LIN {X 0,Y 225.817,Z 674.182,A -85,B 0,C 180,E1 6457.381,E2 6457.381} C_VEL
LIN {X 0,Y 214.23,Z 687.655,A -85,B 0,C 180,E1 6455.161,E2 6455.161} C_VEL
LIN {X 0,Y 203.462,Z 699.057,A -85,B 0,C 180,E1 6452.795,E2 6452.795} C_VEL
LIN {X 0,Y 192.684,Z 709.547,A -85,B 0,C 180,E1 6450.053,E2 6450.053} C_VEL
LIN {X 0,Y 181.69,Z 719.435,A -85,B 0,C 180,E1 6446.76,E2 6446.76} C_VEL
LIN {X 0,Y 170.711,Z 728.616,A -85,B 0,C 180,E1 6442.794,E2 6442.794} C_VEL
LIN {X 0,Y 158.871,Z 737.935,A -85,B 0,C 180,E1 6437.414,E2 6437.414} C_VEL
LIN {X 0,Y 147.139,Z 746.59,A -85,B 0,C 180,E1 6430.202,E2 6430.202} C_VEL
LIN {X 0,Y 139.422,Z 752.214,A -85,B 0,C 180,E1 6423.514,E2 6423.514} C_VEL
LIN {X 0,Y 133.904,Z 756.398,A -85,B 0,C 180,E1 6416.613,E2 6416.613} C_VEL
LIN {X 0,Y 130.17,Z 759.571,A -85,B 0,C 180,E1 6409.122,E2 6409.122} C_VEL
LIN {X 0,Y 128.361,Z 761.606,A -85,B 0,C 180,E1 6401.683,E2 6401.683} C_VEL
LIN {X 0,Y 127.961,Z 762.61,A -85,B 0,C 180,E1 6394.93,E2 6394.93} C_VEL
LIN {X 0,Y 128.002,Z 762.852,A -85,B 0,C 180,E1 6388.657,E2 6388.657} C_VEL
LIN {X 0,Y 128.093,Z 762.147,A -85,B 0,C 180,E1 6381.019,E2 6381.019} C_VEL
LIN {X 0,Y 129.629,Z 760.118,A -85,B 0,C 180,E1 6372.495,E2 6372.495} C_VEL
LIN {X 0,Y 129.83,Z 759.905,A -85,B 0,C 180,E1 6371.863,E2 6371.863} C_VEL
LIN {X 0,Y 130.126,Z 758.8,A -85,B 0,C 180,E1 6368.482,E2 6368.482} C_VEL
LIN {X 0,Y 129.362,Z 754.834,A -85,B 0,C 180,E1 6358.995,E2 6358.995} C_VEL
LIN {X 0,Y 130.84,Z 753.309,A -85,B 0,C 180,E1 6356.462,E2 6356.462} C_VEL
LIN {X 0,Y 138.498,Z 748.084,A -85,B 0,C 180,E1 6349.483,E2 6349.483} C_VEL
LIN {X 0,Y 147.503,Z 741.893,A -85,B 0,C 180,E1 6343.512,E2 6343.512} C_VEL
LIN {X 0,Y 157.231,Z 734.942,A -85,B 0,C 180,E1 6338.547,E2 6338.547} C_VEL
LIN {X 0,Y 167.979,Z 726.812,A -85,B 0,C 180,E1 6334.18,E2 6334.18} C_VEL
LIN {X 0,Y 179.579,Z 717.4,A -85,B 0,C 180,E1 6330.354,E2 6330.354} C_VEL
LIN {X 0,Y 194.261,Z 704.416,A -85,B 0,C 180,E1 6326.43,E2 6326.43} C_VEL
LIN {X 0,Y 208.067,Z 690.555,A -85,B 0,C 180,E1 6323.401,E2 6323.401} C_VEL
LIN {X 0,Y 219.406,Z 677.998,A -85,B 0,C 180,E1 6321.278,E2 6321.278} C_VEL
LIN {X 0,Y 230.156,Z 664.84,A -85,B 0,C 180,E1 6319.506,E2 6319.506} C_VEL
LIN {X 0,Y 240.236,Z 651.143,A -85,B 0,C 180,E1 6318.026,E2 6318.026} C_VEL
LIN {X 0,Y 249.892,Z 636.482,A -85,B 0,C 180,E1 6316.744,E2 6316.744} C_VEL
LIN {X 0,Y 260.396,Z 618.414,A -85,B 0,C 180,E1 6315.489,E2 6315.489} C_VEL
LIN {X 0,Y 270.426,Z 597.812,A -85,B 0,C 180,E1 6314.396,E2 6314.396} C_VEL
LIN {X 0,Y 277.33,Z 581.05,A -85,B 0,C 180,E1 6313.706,E2 6313.706} C_VEL
LIN {X 0,Y 283.119,Z 564.422,A -85,B 0,C 180,E1 6313.162,E2 6313.162} C_VEL
LIN {X 0,Y 288.085,Z 547.062,A -85,B 0,C 180,E1 6312.718,E2 6312.718} C_VEL
LIN {X 0,Y 292.005,Z 529.565,A -85,B 0,C 180,E1 6312.361,E2 6312.361} C_VEL
LIN {X 0,Y 294.954,Z 511.261,A -85,B 0,C 180,E1 6312.045,E2 6312.045} C_VEL
LIN {X 0,Y 303.683,Z 432.891,A -85,B 0,C 180,E1 6310.873,E2 6310.873} C_VEL
LIN {X 0,Y 301.535,Z 427.301,A -85,B 0,C 180,E1 6307.622,E2 6307.622} C_VEL
LIN {X 0,Y 300.202,Z 423.933,A -85,B 0,C 180,E1 6304.585,E2 6304.585} C_VEL
LIN {X 0,Y 299.445,Z 421.761,A -85,B 0,C 180,E1 6299.617,E2 6299.617} C_VEL
LIN {X 0,Y 300.396,Z 424.417,A -85,B 0,C 180,E1 6294.557,E2 6294.557} C_VEL
LIN {X 0,Y 301.941,Z 428.499,A -85,B 0,C 180,E1 6291.334,E2 6291.334} C_VEL
LIN {X 0,Y 303.958,Z 433.602,A -85,B 0,C 180,E1 6288.472,E2 6288.472} C_VEL
LIN {X 0,Y 306.454,Z 440.443,A -85,B 0,C 180,E1 6285.691,E2 6285.691} C_VEL
LIN {X 0,Y 309.329,Z 448.867,A -85,B 0,C 180,E1 6283.039,E2 6283.039} C_VEL
LIN {X 0,Y 316.914,Z 468.169,A -85,B 0,C 180,E1 6277.801,E2 6277.801} C_VEL
LIN {X 0,Y 327.353,Z 485.396,A -85,B 0,C 180,E1 6272.829,E2 6272.829} C_VEL
LIN {X 0,Y 339.675,Z 500.381,A -85,B 0,C 180,E1 6268.401,E2 6268.401} C_VEL
LIN {X 0,Y 361.119,Z 520.754,A -85,B 0,C 180,E1 6262.322,E2 6262.322} C_VEL
LIN {X 0,Y 383.771,Z 538.59,A -85,B 0,C 180,E1 6257.155,E2 6257.155} C_VEL
LIN {X 0,Y 393.502,Z 546.007,A -85,B 0,C 180,E1 6254.935,E2 6254.935} C_VEL
LIN {X 0,Y 403.779,Z 553.746,A -85,B 0,C 180,E1 6252.443,E2 6252.443} C_VEL
LIN {X 0,Y 413.394,Z 561.034,A -85,B 0,C 180,E1 6249.938,E2 6249.938} C_VEL
LIN {X 0,Y 423.167,Z 568.574,A -85,B 0,C 180,E1 6247.215,E2 6247.215} C_VEL
LIN {X 0,Y 430.163,Z 573.895,A -85,B 0,C 180,E1 6245.166,E2 6245.166} C_VEL
LIN {X 0,Y 438.79,Z 580.22,A -85,B 0,C 180,E1 6242.527,E2 6242.527} C_VEL
LIN {X 0,Y 446.99,Z 586.446,A -85,B 0,C 180,E1 6239.78,E2 6239.78} C_VEL
LIN {X 0,Y 453.825,Z 591.043,A -85,B 0,C 180,E1 6237.388,E2 6237.388} C_VEL
LIN {X 0,Y 460.622,Z 596.321,A -85,B 0,C 180,E1 6234.765,E2 6234.765} C_VEL
LIN {X 0,Y 467.284,Z 600.659,A -85,B 0,C 180,E1 6231.988,E2 6231.988} C_VEL
LIN {X 0,Y 471.291,Z 603.671,A -85,B 0,C 180,E1 6230.1,E2 6230.1} C_VEL
LIN {X 0,Y 476.325,Z 607.46,A -85,B 0,C 180,E1 6227.466,E2 6227.466} C_VEL
LIN {X 0,Y 480.91,Z 610.202,A -85,B 0,C 180,E1 6224.802,E2 6224.802} C_VEL
LIN {X 0,Y 484.657,Z 612.219,A -85,B 0,C 180,E1 6222.267,E2 6222.267} C_VEL
LIN {X 0,Y 487.465,Z 614.83,A -85,B 0,C 180,E1 6219.682,E2 6219.682} C_VEL
LIN {X 0,Y 489.719,Z 616.73,A -85,B 0,C 180,E1 6217.036,E2 6217.036} C_VEL
LIN {X 0,Y 491.268,Z 617.837,A -85,B 0,C 180,E1 6214.435,E2 6214.435} C_VEL
LIN {X 0,Y 492.185,Z 618.418,A -85,B 0,C 180,E1 6211.779,E2 6211.779} C_VEL
LIN {X 0,Y 492.284,Z 618.462,A -85,B 0,C 180,E1 6209.302,E2 6209.302} C_VEL
LIN {X 0,Y 491.761,Z 618.158,A -85,B 0,C 180,E1 6206.706,E2 6206.706} C_VEL
LIN {X 0,Y 490.502,Z 617.291,A -85,B 0,C 180,E1 6204.151,E2 6204.151} C_VEL
LIN {X 0,Y 488.442,Z 615.733,A -85,B 0,C 180,E1 6201.399,E2 6201.399} C_VEL
LIN {X 0,Y 485.933,Z 613.485,A -85,B 0,C 180,E1 6198.849,E2 6198.849} C_VEL
LIN {X 0,Y 483.548,Z 611.506,A -85,B 0,C 180,E1 6196.893,E2 6196.893} C_VEL
LIN {X 0,Y 479.591,Z 609.49,A -85,B 0,C 180,E1 6194.4,E2 6194.4} C_VEL
LIN {X 0,Y 474.776,Z 606.383,A -85,B 0,C 180,E1 6191.714,E2 6191.714} C_VEL
LIN {X 0,Y 469.767,Z 602.368,A -85,B 0,C 180,E1 6189.133,E2 6189.133} C_VEL
LIN {X 0,Y 464.002,Z 598.659,A -85,B 0,C 180,E1 6186.636,E2 6186.636} C_VEL
LIN {X 0,Y 457.84,Z 594.204,A -85,B 0,C 180,E1 6184.129,E2 6184.129} C_VEL
LIN {X 0,Y 452.424,Z 590.187,A -85,B 0,C 180,E1 6182.133,E2 6182.133} C_VEL
LIN {X 0,Y 445.952,Z 585.668,A -85,B 0,C 180,E1 6179.856,E2 6179.856} C_VEL
LIN {X 0,Y 438.303,Z 579.905,A -85,B 0,C 180,E1 6177.33,E2 6177.33} C_VEL
LIN {X 0,Y 430.019,Z 573.781,A -85,B 0,C 180,E1 6174.79,E2 6174.79} C_VEL
LIN {X 0,Y 422.676,Z 568.214,A -85,B 0,C 180,E1 6172.641,E2 6172.641} C_VEL
LIN {X 0,Y 412.652,Z 560.525,A -85,B 0,C 180,E1 6169.875,E2 6169.875} C_VEL
LIN {X 0,Y 403.258,Z 553.328,A -85,B 0,C 180,E1 6167.428,E2 6167.428} C_VEL
LIN {X 0,Y 392.511,Z 545.225,A -85,B 0,C 180,E1 6164.83,E2 6164.83} C_VEL
LIN {X 0,Y 382.505,Z 537.63,A -85,B 0,C 180,E1 6162.562,E2 6162.562} C_VEL
LIN {X 0,Y 358.465,Z 518.462,A -85,B 0,C 180,E1 6156.999,E2 6156.999} C_VEL
LIN {X 0,Y 337.709,Z 498.182,A -85,B 0,C 180,E1 6150.96,E2 6150.96} C_VEL
LIN {X 0,Y 325.984,Z 483.515,A -85,B 0,C 180,E1 6146.604,E2 6146.604} C_VEL
LIN {X 0,Y 315.507,Z 465.154,A -85,B 0,C 180,E1 6141.374,E2 6141.374} C_VEL
LIN {X 0,Y 307.789,Z 444.262,A -85,B 0,C 180,E1 6135.594,E2 6135.594} C_VEL
LIN {X 0,Y 304.86,Z 435.971,A -85,B 0,C 180,E1 6132.598,E2 6132.598} C_VEL
LIN {X 0,Y 302.482,Z 429.806,A -85,B 0,C 180,E1 6129.514,E2 6129.514} C_VEL
LIN {X 0,Y 301.107,Z 426.479,A -85,B 0,C 180,E1 6127.153,E2 6127.153} C_VEL
LIN {X 0,Y 300.159,Z 423.881,A -85,B 0,C 180,E1 6124.777,E2 6124.777} C_VEL
LIN {X 0,Y 299.447,Z 421.735,A -85,B 0,C 180,E1 6120,E2 6120} C_VEL
LIN {X 0,Y 300.405,Z 424.423,A -85,B 0,C 180,E1 6114.844,E2 6114.844} C_VEL
LIN {X 0,Y 301.897,Z 428.384,A -85,B 0,C 180,E1 6111.716,E2 6111.716} C_VEL
LIN {X 0,Y 303.703,Z 432.989,A -85,B 0,C 180,E1 6109.095,E2 6109.095} C_VEL
LIN {X 0,Y 294.265,Z 516.426,A -85,B 0,C 180,E1 6107.873,E2 6107.873} C_VEL
LIN {X 0,Y 289.898,Z 539.96,A -85,B 0,C 180,E1 6107.438,E2 6107.438} C_VEL
LIN {X 0,Y 284.283,Z 560.709,A -85,B 0,C 180,E1 6106.941,E2 6106.941} C_VEL
LIN {X 0,Y 278.714,Z 577.321,A -85,B 0,C 180,E1 6106.429,E2 6106.429} C_VEL
LIN {X 0,Y 272.26,Z 593.566,A -85,B 0,C 180,E1 6105.794,E2 6105.794} C_VEL
LIN {X 0,Y 264.94,Z 609.422,A -85,B 0,C 180,E1 6105.02,E2 6105.02} C_VEL
LIN {X 0,Y 256.772,Z 624.857,A -85,B 0,C 180,E1 6104.092,E2 6104.092} C_VEL
LIN {X 0,Y 247.786,Z 639.83,A -85,B 0,C 180,E1 6102.986,E2 6102.986} C_VEL
LIN {X 0,Y 237.153,Z 655.552,A -85,B 0,C 180,E1 6101.535,E2 6101.535} C_VEL
LIN {X 0,Y 222.822,Z 674.005,A -85,B 0,C 180,E1 6099.308,E2 6099.308} C_VEL
LIN {X 0,Y 211.394,Z 686.997,A -85,B 0,C 180,E1 6097.253,E2 6097.253} C_VEL
LIN {X 0,Y 199.871,Z 698.879,A -85,B 0,C 180,E1 6094.872,E2 6094.872} C_VEL
LIN {X 0,Y 188.745,Z 709.369,A -85,B 0,C 180,E1 6092.199,E2 6092.199} C_VEL
LIN {X 0,Y 177.345,Z 719.257,A -85,B 0,C 180,E1 6088.967,E2 6088.967} C_VEL
LIN {X 0,Y 166.079,Z 728.293,A -85,B 0,C 180,E1 6085.113,E2 6085.113} C_VEL
LIN {X 0,Y 154.39,Z 737.049,A -85,B 0,C 180,E1 6080.121,E2 6080.121} C_VEL
LIN {X 0,Y 141.499,Z 746.082,A -85,B 0,C 180,E1 6072.7,E2 6072.7} C_VEL
LIN {X 0,Y 132.688,Z 752.036,A -85,B 0,C 180,E1 6065.462,E2 6065.462} C_VEL
LIN {X 0,Y 126.667,Z 756.22,A -85,B 0,C 180,E1 6058.266,E2 6058.266} C_VEL
LIN {X 0,Y 122.584,Z 759.342,A -85,B 0,C 180,E1 6050.53,E2 6050.53} C_VEL
LIN {X 0,Y 120.454,Z 761.429,A -85,B 0,C 180,E1 6042.462,E2 6042.462} C_VEL
LIN {X 0,Y 119.963,Z 762.434,A -85,B 0,C 180,E1 6035.26,E2 6035.26} C_VEL
LIN {X 0,Y 120.001,Z 762.677,A -85,B 0,C 180,E1 6028.568,E2 6028.568} C_VEL
LIN {X 0,Y 120.132,Z 761.97,A -85,B 0,C 180,E1 6020.419,E2 6020.419} C_VEL
LIN {X 0,Y 121.918,Z 759.933,A -85,B 0,C 180,E1 6011.324,E2 6011.324} C_VEL
LIN {X 0,Y 125.803,Z 756.85,A -85,B 0,C 180,E1 6003.065,E2 6003.065} C_VEL
LIN {X 0,Y 130.84,Z 753.309,A -85,B 0,C 180,E1 5996.462,E2 5996.462} C_VEL
LIN {X 0,Y 132.864,Z 751.373,A -85,B 0,C 180,E1 5993.316,E2 5993.316} C_VEL
LIN {X 0,Y 136.774,Z 745.591,A -85,B 0,C 180,E1 5984.772,E2 5984.772} C_VEL
LIN {X 0,Y 139.622,Z 743.303,A -85,B 0,C 180,E1 5982.461,E2 5982.461} C_VEL
LIN {X 0,Y 150.928,Z 735.701,A -85,B 0,C 180,E1 5976.725,E2 5976.725} C_VEL
LIN {X 0,Y 162.074,Z 727.717,A -85,B 0,C 180,E1 5972.319,E2 5972.319} C_VEL
LIN {X 0,Y 173.278,Z 719.078,A -85,B 0,C 180,E1 5968.719,E2 5968.719} C_VEL
LIN {X 0,Y 185.083,Z 709.19,A -85,B 0,C 180,E1 5965.568,E2 5965.568} C_VEL
LIN {X 0,Y 196.552,Z 698.7,A -85,B 0,C 180,E1 5962.979,E2 5962.979} C_VEL
LIN {X 0,Y 208.386,Z 686.819,A -85,B 0,C 180,E1 5960.686,E2 5960.686} C_VEL
LIN {X 0,Y 222.605,Z 670.953,A -85,B 0,C 180,E1 5958.326,E2 5958.326} C_VEL
LIN {X 0,Y 235.611,Z 654.115,A -85,B 0,C 180,E1 5956.469,E2 5956.469} C_VEL
LIN {X 0,Y 245.822,Z 639.217,A -85,B 0,C 180,E1 5955.177,E2 5955.177} C_VEL
LIN {X 0,Y 254.679,Z 624.68,A -85,B 0,C 180,E1 5954.162,E2 5954.162} C_VEL
LIN {X 0,Y 262.974,Z 609.246,A -85,B 0,C 180,E1 5953.285,E2 5953.285} C_VEL
LIN {X 0,Y 270.399,Z 593.389,A -85,B 0,C 180,E1 5952.554,E2 5952.554} C_VEL
LIN {X 0,Y 277.407,Z 575.902,A -85,B 0,C 180,E1 5951.913,E2 5951.913} C_VEL
LIN {X 0,Y 284.639,Z 553.835,A -85,B 0,C 180,E1 5951.303,E2 5951.303} C_VEL
LIN {X 0,Y 289.757,Z 532.601,A -85,B 0,C 180,E1 5950.873,E2 5950.873} C_VEL
LIN {X 0,Y 292.91,Z 514.474,A -85,B 0,C 180,E1 5950.565,E2 5950.565} C_VEL
LIN {X 0,Y 301.601,Z 438.572,A -85,B 0,C 180,E1 5949.445,E2 5949.445} C_VEL
LIN {X 0,Y 300.034,Z 434.394,A -85,B 0,C 180,E1 5946.698,E2 5946.698} C_VEL
LIN {X 0,Y 299.09,Z 431.72,A -85,B 0,C 180,E1 5944.218,E2 5944.218} C_VEL
LIN {X 0,Y 298.467,Z 429.724,A -85,B 0,C 180,E1 5939.616,E2 5939.616} C_VEL
LIN {X 0,Y 299.335,Z 432.351,A -85,B 0,C 180,E1 5934.729,E2 5934.729} C_VEL
LIN {X 0,Y 300.717,Z 436.195,A -85,B 0,C 180,E1 5931.684,E2 5931.684} C_VEL
LIN {X 0,Y 302.598,Z 441.275,A -85,B 0,C 180,E1 5928.854,E2 5928.854} C_VEL
LIN {X 0,Y 304.806,Z 447.733,A -85,B 0,C 180,E1 5926.241,E2 5926.241} C_VEL
LIN {X 0,Y 307.381,Z 455.777,A -85,B 0,C 180,E1 5923.706,E2 5923.706} C_VEL
LIN {X 0,Y 314.649,Z 475.053,A -85,B 0,C 180,E1 5918.418,E2 5918.418} C_VEL
LIN {X 0,Y 324.896,Z 492.411,A -85,B 0,C 180,E1 5913.349,E2 5913.349} C_VEL
LIN {X 0,Y 335.831,Z 506.221,A -85,B 0,C 180,E1 5909.196,E2 5909.196} C_VEL
LIN {X 0,Y 353.843,Z 524.22,A -85,B 0,C 180,E1 5903.7,E2 5903.7} C_VEL
LIN {X 0,Y 379.885,Z 545.436,A -85,B 0,C 180,E1 5897.382,E2 5897.382} C_VEL
LIN {X 0,Y 389.932,Z 553.073,A -85,B 0,C 180,E1 5895.104,E2 5895.104} C_VEL
LIN {X 0,Y 400.416,Z 560.982,A -85,B 0,C 180,E1 5892.553,E2 5892.553} C_VEL
LIN {X 0,Y 410.613,Z 568.64,A -85,B 0,C 180,E1 5889.909,E2 5889.909} C_VEL
LIN {X 0,Y 419.937,Z 575.857,A -85,B 0,C 180,E1 5887.319,E2 5887.319} C_VEL
LIN {X 0,Y 428.263,Z 582.208,A -85,B 0,C 180,E1 5884.885,E2 5884.885} C_VEL
LIN {X 0,Y 436.186,Z 587.913,A -85,B 0,C 180,E1 5882.435,E2 5882.435} C_VEL
LIN {X 0,Y 443.453,Z 593.466,A -85,B 0,C 180,E1 5880.021,E2 5880.021} C_VEL
LIN {X 0,Y 451.356,Z 598.755,A -85,B 0,C 180,E1 5877.291,E2 5877.291} C_VEL
LIN {X 0,Y 458.099,Z 604.069,A -85,B 0,C 180,E1 5874.635,E2 5874.635} C_VEL
LIN {X 0,Y 464.596,Z 608.228,A -85,B 0,C 180,E1 5871.938,E2 5871.938} C_VEL
LIN {X 0,Y 469.631,Z 612.116,A -85,B 0,C 180,E1 5869.525,E2 5869.525} C_VEL
LIN {X 0,Y 474.534,Z 615.637,A -85,B 0,C 180,E1 5866.902,E2 5866.902} C_VEL
LIN {X 0,Y 479.033,Z 618.174,A -85,B 0,C 180,E1 5864.257,E2 5864.257} C_VEL
LIN {X 0,Y 481.979,Z 619.832,A -85,B 0,C 180,E1 5862.215,E2 5862.215} C_VEL
LIN {X 0,Y 484.771,Z 622.412,A -85,B 0,C 180,E1 5859.616,E2 5859.616} C_VEL
LIN {X 0,Y 486.974,Z 624.267,A -85,B 0,C 180,E1 5856.957,E2 5856.957} C_VEL
LIN {X 0,Y 488.51,Z 625.367,A -85,B 0,C 180,E1 5854.343,E2 5854.343} C_VEL
LIN {X 0,Y 489.414,Z 625.923,A -85,B 0,C 180,E1 5851.756,E2 5851.756} C_VEL
LIN {X 0,Y 489.504,Z 625.963,A -85,B 0,C 180,E1 5849.298,E2 5849.298} C_VEL
LIN {X 0,Y 488.977,Z 625.658,A -85,B 0,C 180,E1 5846.718,E2 5846.718} C_VEL
LIN {X 0,Y 487.707,Z 624.783,A -85,B 0,C 180,E1 5844.117,E2 5844.117} C_VEL
LIN {X 0,Y 485.615,Z 623.208,A -85,B 0,C 180,E1 5841.356,E2 5841.356} C_VEL
LIN {X 0,Y 483.115,Z 620.952,A -85,B 0,C 180,E1 5838.783,E2 5838.783} C_VEL
LIN {X 0,Y 480.795,Z 619.019,A -85,B 0,C 180,E1 5836.9,E2 5836.9} C_VEL
LIN {X 0,Y 476.652,Z 616.906,A -85,B 0,C 180,E1 5834.302,E2 5834.302} C_VEL
LIN {X 0,Y 471.906,Z 613.842,A -85,B 0,C 180,E1 5831.666,E2 5831.666} C_VEL
LIN {X 0,Y 466.751,Z 609.74,A -85,B 0,C 180,E1 5829.041,E2 5829.041} C_VEL
LIN {X 0,Y 460.786,Z 605.909,A -85,B 0,C 180,E1 5826.471,E2 5826.471} C_VEL
LIN {X 0,Y 454.378,Z 601.236,A -85,B 0,C 180,E1 5823.875,E2 5823.875} C_VEL
LIN {X 0,Y 449.746,Z 597.783,A -85,B 0,C 180,E1 5822.172,E2 5822.172} C_VEL
LIN {X 0,Y 443.405,Z 593.433,A -85,B 0,C 180,E1 5819.964,E2 5819.964} C_VEL
LIN {X 0,Y 435.55,Z 587.487,A -85,B 0,C 180,E1 5817.356,E2 5817.356} C_VEL
LIN {X 0,Y 426.629,Z 580.931,A -85,B 0,C 180,E1 5814.633,E2 5814.633} C_VEL
LIN {X 0,Y 419.431,Z 575.498,A -85,B 0,C 180,E1 5812.547,E2 5812.547} C_VEL
LIN {X 0,Y 411.112,Z 568.993,A -85,B 0,C 180,E1 5810.225,E2 5810.225} C_VEL
LIN {X 0,Y 400.943,Z 561.405,A -85,B 0,C 180,E1 5807.577,E2 5807.577} C_VEL
LIN {X 0,Y 390.538,Z 553.549,A -85,B 0,C 180,E1 5805.046,E2 5805.046} C_VEL
LIN {X 0,Y 380.193,Z 545.656,A -85,B 0,C 180,E1 5802.678,E2 5802.678} C_VEL
LIN {X 0,Y 353.714,Z 524.102,A -85,B 0,C 180,E1 5796.265,E2 5796.265} C_VEL
LIN {X 0,Y 335.517,Z 505.836,A -85,B 0,C 180,E1 5790.687,E2 5790.687} C_VEL
LIN {X 0,Y 324.222,Z 491.478,A -85,B 0,C 180,E1 5786.365,E2 5786.365} C_VEL
LIN {X 0,Y 313.71,Z 473.008,A -85,B 0,C 180,E1 5781.013,E2 5781.013} C_VEL
LIN {X 0,Y 305.885,Z 450.998,A -85,B 0,C 180,E1 5774.869,E2 5774.869} C_VEL
LIN {X 0,Y 303.192,Z 442.887,A -85,B 0,C 180,E1 5771.895,E2 5771.895} C_VEL
LIN {X 0,Y 300.993,Z 436.928,A -85,B 0,C 180,E1 5768.79,E2 5768.79} C_VEL
LIN {X 0,Y 299.888,Z 434.067,A -85,B 0,C 180,E1 5766.702,E2 5766.702} C_VEL
LIN {X 0,Y 299.115,Z 431.763,A -85,B 0,C 180,E1 5764.602,E2 5764.602} C_VEL
LIN {X 0,Y 298.47,Z 429.691,A -85,B 0,C 180,E1 5760,E2 5760} C_VEL
LIN {X 0,Y 299.343,Z 432.355,A -85,B 0,C 180,E1 5755.018,E2 5755.018} C_VEL
LIN {X 0,Y 300.674,Z 436.079,A -85,B 0,C 180,E1 5752.067,E2 5752.067} C_VEL
LIN {X 0,Y 301.616,Z 438.808,A -85,B 0,C 180,E1 5750.505,E2 5750.505} C_VEL
LIN {X 0,Y 292.661,Z 516.428,A -85,B 0,C 180,E1 5749.405,E2 5749.405} C_VEL
LIN {X 0,Y 288.175,Z 540.116,A -85,B 0,C 180,E1 5748.987,E2 5748.987} C_VEL
LIN {X 0,Y 282.578,Z 560.533,A -85,B 0,C 180,E1 5748.526,E2 5748.526} C_VEL
LIN {X 0,Y 276.939,Z 577.145,A -85,B 0,C 180,E1 5748.046,E2 5748.046} C_VEL
LIN {X 0,Y 270.399,Z 593.39,A -85,B 0,C 180,E1 5747.446,E2 5747.446} C_VEL
LIN {X 0,Y 262.974,Z 609.246,A -85,B 0,C 180,E1 5746.715,E2 5746.715} C_VEL
LIN {X 0,Y 254.68,Z 624.681,A -85,B 0,C 180,E1 5745.837,E2 5745.837} C_VEL
LIN {X 0,Y 245.543,Z 639.653,A -85,B 0,C 180,E1 5744.789,E2 5744.789} C_VEL
LIN {X 0,Y 234.715,Z 655.375,A -85,B 0,C 180,E1 5743.41,E2 5743.41} C_VEL
LIN {X 0,Y 220.085,Z 673.827,A -85,B 0,C 180,E1 5741.285,E2 5741.285} C_VEL
LIN {X 0,Y 208.386,Z 686.82,A -85,B 0,C 180,E1 5739.314,E2 5739.314} C_VEL
LIN {X 0,Y 196.551,Z 698.701,A -85,B 0,C 180,E1 5737.021,E2 5737.021} C_VEL
LIN {X 0,Y 184.676,Z 709.545,A -85,B 0,C 180,E1 5734.332,E2 5734.332} C_VEL
LIN {X 0,Y 172.511,Z 719.697,A -85,B 0,C 180,E1 5731.055,E2 5731.055} C_VEL
LIN {X 0,Y 159.918,Z 729.342,A -85,B 0,C 180,E1 5726.9,E2 5726.9} C_VEL
LIN {X 0,Y 144.46,Z 740.113,A -85,B 0,C 180,E1 5720.191,E2 5720.191} C_VEL
LIN {X 0,Y 133.974,Z 746.902,A -85,B 0,C 180,E1 5713.947,E2 5713.947} C_VEL
LIN {X 0,Y 125.682,Z 752.128,A -85,B 0,C 180,E1 5707.197,E2 5707.197} C_VEL
LIN {X 0,Y 119.221,Z 756.252,A -85,B 0,C 180,E1 5699.654,E2 5699.654} C_VEL
LIN {X 0,Y 114.804,Z 759.314,A -85,B 0,C 180,E1 5691.454,E2 5691.454} C_VEL
LIN {X 0,Y 112.489,Z 761.343,A -85,B 0,C 180,E1 5682.838,E2 5682.838} C_VEL
LIN {X 0,Y 111.964,Z 762.29,A -85,B 0,C 180,E1 5675.123,E2 5675.123} C_VEL
LIN {X 0,Y 112,Z 762.502,A -85,B 0,C 180,E1 5668.465,E2 5668.465} C_VEL
LIN {X 0,Y 112.184,Z 761.794,A -85,B 0,C 180,E1 5659.733,E2 5659.733} C_VEL
LIN {X 0,Y 114.245,Z 759.763,A -85,B 0,C 180,E1 5650.045,E2 5650.045} C_VEL
LIN {X 0,Y 118.613,Z 756.657,A -85,B 0,C 180,E1 5641.249,E2 5641.249} C_VEL
LIN {X 0,Y 124.82,Z 752.671,A -85,B 0,C 180,E1 5633.651,E2 5633.651} C_VEL
LIN {X 0,Y 132.911,Z 747.571,A -85,B 0,C 180,E1 5626.804,E2 5626.804} C_VEL
LIN {X 0,Y 139.622,Z 743.303,A -85,B 0,C 180,E1 5622.461,E2 5622.461} C_VEL
LIN {X 0,Y 143.09,Z 740.557,A -85,B 0,C 180,E1 5619.872,E2 5619.872} C_VEL
LIN {X 0,Y 150.268,Z 733.366,A -85,B 0,C 180,E1 5613.073,E2 5613.073} C_VEL
LIN {X 0,Y 154.478,Z 729.986,A -85,B 0,C 180,E1 5610.975,E2 5610.975} C_VEL
LIN {X 0,Y 167.92,Z 720.137,A -85,B 0,C 180,E1 5606.739,E2 5606.739} C_VEL
LIN {X 0,Y 180.885,Z 709.713,A -85,B 0,C 180,E1 5603.439,E2 5603.439} C_VEL
LIN {X 0,Y 192.665,Z 699.314,A -85,B 0,C 180,E1 5600.927,E2 5600.927} C_VEL
LIN {X 0,Y 203.904,Z 688.42,A -85,B 0,C 180,E1 5598.864,E2 5598.864} C_VEL
LIN {X 0,Y 215.623,Z 675.879,A -85,B 0,C 180,E1 5596.987,E2 5596.987} C_VEL
LIN {X 0,Y 227.078,Z 662.245,A -85,B 0,C 180,E1 5595.38,E2 5595.38} C_VEL
LIN {X 0,Y 240.328,Z 644.448,A -85,B 0,C 180,E1 5593.748,E2 5593.748} C_VEL
LIN {X 0,Y 251.896,Z 626.115,A -85,B 0,C 180,E1 5592.485,E2 5592.485} C_VEL
LIN {X 0,Y 260.772,Z 609.99,A -85,B 0,C 180,E1 5591.61,E2 5591.61} C_VEL
LIN {X 0,Y 268.294,Z 594.275,A -85,B 0,C 180,E1 5590.921,E2 5590.921} C_VEL
LIN {X 0,Y 274.913,Z 578.212,A -85,B 0,C 180,E1 5590.358,E2 5590.358} C_VEL
LIN {X 0,Y 280.616,Z 561.843,A -85,B 0,C 180,E1 5589.906,E2 5589.906} C_VEL
LIN {X 0,Y 285.677,Z 544.056,A -85,B 0,C 180,E1 5589.52,E2 5589.52} C_VEL
LIN {X 0,Y 290.482,Z 521.745,A -85,B 0,C 180,E1 5589.127,E2 5589.127} C_VEL
LIN {X 0,Y 294.809,Z 487.75,A -85,B 0,C 180,E1 5588.645,E2 5588.645} C_VEL
LIN {X 0,Y 299.72,Z 444.504,A -85,B 0,C 180,E1 5588.055,E2 5588.055} C_VEL
LIN {X 0,Y 298.696,Z 441.659,A -85,B 0,C 180,E1 5585.957,E2 5585.957} C_VEL
LIN {X 0,Y 298.05,Z 439.601,A -85,B 0,C 180,E1 5584.04,E2 5584.04} C_VEL
LIN {X 0,Y 297.489,Z 437.69,A -85,B 0,C 180,E1 5579.615,E2 5579.615} C_VEL
LIN {X 0,Y 298.25,Z 440.161,A -85,B 0,C 180,E1 5574.999,E2 5574.999} C_VEL
LIN {X 0,Y 299.554,Z 444.038,A -85,B 0,C 180,E1 5571.941,E2 5571.941} C_VEL
LIN {X 0,Y 301.458,Z 449.556,A -85,B 0,C 180,E1 5568.957,E2 5568.957} C_VEL
LIN {X 0,Y 303.516,Z 456.1,A -85,B 0,C 180,E1 5566.425,E2 5566.425} C_VEL
LIN {X 0,Y 305.808,Z 463.874,A -85,B 0,C 180,E1 5564.059,E2 5564.059} C_VEL
LIN {X 0,Y 312.923,Z 483.011,A -85,B 0,C 180,E1 5558.736,E2 5558.736} C_VEL
LIN {X 0,Y 323.889,Z 501.543,A -85,B 0,C 180,E1 5553.259,E2 5553.259} C_VEL
LIN {X 0,Y 338.433,Z 519.223,A -85,B 0,C 180,E1 5547.772,E2 5547.772} C_VEL
LIN {X 0,Y 357.634,Z 537.531,A -85,B 0,C 180,E1 5542.042,E2 5542.042} C_VEL
LIN {X 0,Y 380.681,Z 555.751,A -85,B 0,C 180,E1 5536.515,E2 5536.515} C_VEL
LIN {X 0,Y 391.612,Z 564.172,A -85,B 0,C 180,E1 5533.944,E2 5533.944} C_VEL
LIN {X 0,Y 401.536,Z 571.781,A -85,B 0,C 180,E1 5531.449,E2 5531.449} C_VEL
LIN {X 0,Y 410.626,Z 578.592,A -85,B 0,C 180,E1 5529.033,E2 5529.033} C_VEL
LIN {X 0,Y 419.479,Z 585.163,A -85,B 0,C 180,E1 5526.554,E2 5526.554} C_VEL
LIN {X 0,Y 428.549,Z 592.2,A -85,B 0,C 180,E1 5523.837,E2 5523.837} C_VEL
LIN {X 0,Y 436.065,Z 597.592,A -85,B 0,C 180,E1 5521.461,E2 5521.461} C_VEL
LIN {X 0,Y 442.945,Z 602.736,A -85,B 0,C 180,E1 5519.12,E2 5519.12} C_VEL
LIN {X 0,Y 449.61,Z 607.3,A -85,B 0,C 180,E1 5516.774,E2 5516.774} C_VEL
LIN {X 0,Y 456.445,Z 612.475,A -85,B 0,C 180,E1 5514.041,E2 5514.041} C_VEL
LIN {X 0,Y 463.052,Z 616.623,A -85,B 0,C 180,E1 5511.267,E2 5511.267} C_VEL
LIN {X 0,Y 468.396,Z 620.937,A -85,B 0,C 180,E1 5508.544,E2 5508.544} C_VEL
LIN {X 0,Y 473.356,Z 624.177,A -85,B 0,C 180,E1 5505.81,E2 5505.81} C_VEL
LIN {X 0,Y 477.617,Z 626.357,A -85,B 0,C 180,E1 5503.189,E2 5503.189} C_VEL
LIN {X 0,Y 479.81,Z 628.141,A -85,B 0,C 180,E1 5501.417,E2 5501.417} C_VEL
LIN {X 0,Y 482.399,Z 630.472,A -85,B 0,C 180,E1 5498.822,E2 5498.822} C_VEL
LIN {X 0,Y 484.472,Z 632.055,A -85,B 0,C 180,E1 5496.16,E2 5496.16} C_VEL
LIN {X 0,Y 485.834,Z 633.014,A -85,B 0,C 180,E1 5493.46,E2 5493.46} C_VEL
LIN {X 0,Y 486.4,Z 633.343,A -85,B 0,C 180,E1 5490.942,E2 5490.942} C_VEL
LIN {X 0,Y 486.324,Z 633.313,A -85,B 0,C 180,E1 5488.351,E2 5488.351} C_VEL
LIN {X 0,Y 485.442,Z 632.747,A -85,B 0,C 180,E1 5485.63,E2 5485.63} C_VEL
LIN {X 0,Y 483.881,Z 631.639,A -85,B 0,C 180,E1 5482.998,E2 5482.998} C_VEL
LIN {X 0,Y 481.607,Z 629.742,A -85,B 0,C 180,E1 5480.32,E2 5480.32} C_VEL
LIN {X 0,Y 478.826,Z 627.154,A -85,B 0,C 180,E1 5477.704,E2 5477.704} C_VEL
LIN {X 0,Y 475.145,Z 625.14,A -85,B 0,C 180,E1 5475.25,E2 5475.25} C_VEL
LIN {X 0,Y 470.438,Z 622.377,A -85,B 0,C 180,E1 5472.564,E2 5472.564} C_VEL
LIN {X 0,Y 465.099,Z 618.372,A -85,B 0,C 180,E1 5469.752,E2 5469.752} C_VEL
LIN {X 0,Y 461.325,Z 615.512,A -85,B 0,C 180,E1 5467.981,E2 5467.981} C_VEL
LIN {X 0,Y 454.716,Z 611.271,A -85,B 0,C 180,E1 5465.253,E2 5465.253} C_VEL
LIN {X 0,Y 448.032,Z 606.006,A -85,B 0,C 180,E1 5462.634,E2 5462.634} C_VEL
LIN {X 0,Y 439.737,Z 600.437,A -85,B 0,C 180,E1 5459.776,E2 5459.776} C_VEL
LIN {X 0,Y 432.331,Z 594.826,A -85,B 0,C 180,E1 5457.337,E2 5457.337} C_VEL
LIN {X 0,Y 423.676,Z 588.509,A -85,B 0,C 180,E1 5454.681,E2 5454.681} C_VEL
LIN {X 0,Y 415.058,Z 582.011,A -85,B 0,C 180,E1 5452.201,E2 5452.201} C_VEL
LIN {X 0,Y 406.119,Z 575.128,A -85,B 0,C 180,E1 5449.751,E2 5449.751} C_VEL
LIN {X 0,Y 396.371,Z 567.744,A -85,B 0,C 180,E1 5447.23,E2 5447.23} C_VEL
LIN {X 0,Y 385.645,Z 559.667,A -85,B 0,C 180,E1 5444.64,E2 5444.64} C_VEL
LIN {X 0,Y 376.001,Z 552.329,A -85,B 0,C 180,E1 5442.438,E2 5442.438} C_VEL
LIN {X 0,Y 351.631,Z 532.3,A -85,B 0,C 180,E1 5436.312,E2 5436.312} C_VEL
LIN {X 0,Y 332.627,Z 512.698,A -85,B 0,C 180,E1 5430.183,E2 5430.183} C_VEL
LIN {X 0,Y 321.436,Z 497.955,A -85,B 0,C 180,E1 5425.669,E2 5425.669} C_VEL
LIN {X 0,Y 311.111,Z 478.937,A -85,B 0,C 180,E1 5420.114,E2 5420.114} C_VEL
LIN {X 0,Y 304.032,Z 457.731,A -85,B 0,C 180,E1 5414.134,E2 5414.134} C_VEL
LIN {X 0,Y 301.637,Z 450.053,A -85,B 0,C 180,E1 5411.278,E2 5411.278} C_VEL
LIN {X 0,Y 299.605,Z 444.184,A -85,B 0,C 180,E1 5408.154,E2 5408.154} C_VEL
LIN {X 0,Y 298.535,Z 441.209,A -85,B 0,C 180,E1 5405.863,E2 5405.863} C_VEL
LIN {X 0,Y 298.013,Z 439.549,A -85,B 0,C 180,E1 5404.233,E2 5404.233} C_VEL
LIN {X 0,Y 297.493,Z 437.65,A -85,B 0,C 180,E1 5400,E2 5400} C_VEL
LIN {X 0,Y 298.257,Z 440.165,A -85,B 0,C 180,E1 5395.289,E2 5395.289} C_VEL
LIN {X 0,Y 299.512,Z 443.922,A -85,B 0,C 180,E1 5392.326,E2 5392.326} C_VEL
LIN {X 0,Y 299.699,Z 444.754,A -85,B 0,C 180,E1 5391.933,E2 5391.933} C_VEL
LIN {X 0,Y 291.267,Z 516.442,A -85,B 0,C 180,E1 5390.953,E2 5390.953} C_VEL
LIN {X 0,Y 286.632,Z 540.398,A -85,B 0,C 180,E1 5390.551,E2 5390.551} C_VEL
LIN {X 0,Y 281.092,Z 560.358,A -85,B 0,C 180,E1 5390.129,E2 5390.129} C_VEL
LIN {X 0,Y 275.387,Z 576.97,A -85,B 0,C 180,E1 5389.681,E2 5389.681} C_VEL
LIN {X 0,Y 268.766,Z 593.214,A -85,B 0,C 180,E1 5389.12,E2 5389.12} C_VEL
LIN {X 0,Y 261.241,Z 609.07,A -85,B 0,C 180,E1 5388.434,E2 5388.434} C_VEL
LIN {X 0,Y 252.827,Z 624.505,A -85,B 0,C 180,E1 5387.61,E2 5387.61} C_VEL
LIN {X 0,Y 243.548,Z 639.477,A -85,B 0,C 180,E1 5386.624,E2 5386.624} C_VEL
LIN {X 0,Y 232.242,Z 655.6,A -85,B 0,C 180,E1 5385.284,E2 5385.284} C_VEL
LIN {X 0,Y 217.618,Z 673.65,A -85,B 0,C 180,E1 5383.308,E2 5383.308} C_VEL
LIN {X 0,Y 205.655,Z 686.642,A -85,B 0,C 180,E1 5381.433,E2 5381.433} C_VEL
LIN {X 0,Y 193.519,Z 698.523,A -85,B 0,C 180,E1 5379.241,E2 5379.241} C_VEL
LIN {X 0,Y 181.713,Z 709.012,A -85,B 0,C 180,E1 5376.751,E2 5376.751} C_VEL
LIN {X 0,Y 169.507,Z 718.9,A -85,B 0,C 180,E1 5373.701,E2 5373.701} C_VEL
LIN {X 0,Y 157.102,Z 728.08,A -85,B 0,C 180,E1 5369.936,E2 5369.936} C_VEL
LIN {X 0,Y 143.358,Z 737.436,A -85,B 0,C 180,E1 5364.626,E2 5364.626} C_VEL
LIN {X 0,Y 129.372,Z 746.054,A -85,B 0,C 180,E1 5357.234,E2 5357.234} C_VEL
LIN {X 0,Y 119.75,Z 751.678,A -85,B 0,C 180,E1 5350.004,E2 5350.004} C_VEL
LIN {X 0,Y 112.564,Z 755.863,A -85,B 0,C 180,E1 5342.201,E2 5342.201} C_VEL
LIN {X 0,Y 107.506,Z 758.986,A -85,B 0,C 180,E1 5333.57,E2 5333.57} C_VEL
LIN {X 0,Y 104.713,Z 761.076,A -85,B 0,C 180,E1 5324.373,E2 5324.373} C_VEL
LIN {X 0,Y 103.978,Z 762.083,A -85,B 0,C 180,E1 5316.071,E2 5316.071} C_VEL
LIN {X 0,Y 104.01,Z 762.355,A -85,B 0,C 180,E1 5308.87,E2 5308.87} C_VEL
LIN {X 0,Y 104.197,Z 761.708,A -85,B 0,C 180,E1 5299.496,E2 5299.496} C_VEL
LIN {X 0,Y 106.644,Z 759.585,A -85,B 0,C 180,E1 5288.555,E2 5288.555} C_VEL
LIN {X 0,Y 111.51,Z 756.493,A -85,B 0,C 180,E1 5279.267,E2 5279.267} C_VEL
LIN {X 0,Y 118.338,Z 752.492,A -85,B 0,C 180,E1 5271.305,E2 5271.305} C_VEL
LIN {X 0,Y 127.072,Z 747.392,A -85,B 0,C 180,E1 5264.279,E2 5264.279} C_VEL
LIN {X 0,Y 137.4,Z 741.135,A -85,B 0,C 180,E1 5258.202,E2 5258.202} C_VEL
LIN {X 0,Y 149.021,Z 733.647,A -85,B 0,C 180,E1 5253.007,E2 5253.007} C_VEL
LIN {X 0,Y 154.478,Z 729.986,A -85,B 0,C 180,E1 5250.975,E2 5250.975} C_VEL
LIN {X 0,Y 158.847,Z 726.473,A -85,B 0,C 180,E1 5249.006,E2 5249.006} C_VEL
LIN {X 0,Y 168.347,Z 717.551,A -85,B 0,C 180,E1 5243.627,E2 5243.627} C_VEL
LIN {X 0,Y 173.066,Z 713.456,A -85,B 0,C 180,E1 5242.084,E2 5242.084} C_VEL
LIN {X 0,Y 188.161,Z 700.718,A -85,B 0,C 180,E1 5238.957,E2 5238.957} C_VEL
LIN {X 0,Y 200.635,Z 689.027,A -85,B 0,C 180,E1 5236.801,E2 5236.801} C_VEL
LIN {X 0,Y 212.242,Z 676.966,A -85,B 0,C 180,E1 5235.063,E2 5235.063} C_VEL
LIN {X 0,Y 223.221,Z 664.309,A -85,B 0,C 180,E1 5233.618,E2 5233.618} C_VEL
LIN {X 0,Y 233.915,Z 650.55,A -85,B 0,C 180,E1 5232.36,E2 5232.36} C_VEL
LIN {X 0,Y 244.153,Z 635.748,A -85,B 0,C 180,E1 5231.275,E2 5231.275} C_VEL
LIN {X 0,Y 255.479,Z 617.08,A -85,B 0,C 180,E1 5230.204,E2 5230.204} C_VEL
LIN {X 0,Y 265.457,Z 597.284,A -85,B 0,C 180,E1 5229.343,E2 5229.343} C_VEL
LIN {X 0,Y 272.626,Z 580.523,A -85,B 0,C 180,E1 5228.777,E2 5228.777} C_VEL
LIN {X 0,Y 278.625,Z 563.896,A -85,B 0,C 180,E1 5228.336,E2 5228.336} C_VEL
LIN {X 0,Y 283.759,Z 546.544,A -85,B 0,C 180,E1 5227.975,E2 5227.975} C_VEL
LIN {X 0,Y 287.792,Z 529.155,A -85,B 0,C 180,E1 5227.679,E2 5227.679} C_VEL
LIN {X 0,Y 290.857,Z 510.941,A -85,B 0,C 180,E1 5227.409,E2 5227.409} C_VEL
LIN {X 0,Y 297.986,Z 450.482,A -85,B 0,C 180,E1 5226.604,E2 5226.604} C_VEL
LIN {X 0,Y 297.013,Z 447.483,A -85,B 0,C 180,E1 5223.861,E2 5223.861} C_VEL
LIN {X 0,Y 296.51,Z 445.66,A -85,B 0,C 180,E1 5219.614,E2 5219.614} C_VEL
LIN {X 0,Y 297.171,Z 447.971,A -85,B 0,C 180,E1 5215.272,E2 5215.272} C_VEL
LIN {X 0,Y 298.349,Z 451.732,A -85,B 0,C 180,E1 5212.296,E2 5212.296} C_VEL
LIN {X 0,Y 300.218,Z 457.515,A -85,B 0,C 180,E1 5209.202,E2 5209.202} C_VEL
LIN {X 0,Y 302.515,Z 465.463,A -85,B 0,C 180,E1 5206.282,E2 5206.282} C_VEL
LIN {X 0,Y 310.925,Z 490.348,A -85,B 0,C 180,E1 5199.234,E2 5199.234} C_VEL
LIN {X 0,Y 320.466,Z 507.275,A -85,B 0,C 180,E1 5194.149,E2 5194.149} C_VEL
LIN {X 0,Y 331.055,Z 521.373,A -85,B 0,C 180,E1 5189.734,E2 5189.734} C_VEL
LIN {X 0,Y 349.886,Z 540.881,A -85,B 0,C 180,E1 5183.478,E2 5183.478} C_VEL
LIN {X 0,Y 374.602,Z 561.138,A -85,B 0,C 180,E1 5177.106,E2 5177.106} C_VEL
LIN {X 0,Y 385.705,Z 569.643,A -85,B 0,C 180,E1 5174.528,E2 5174.528} C_VEL
LIN {X 0,Y 394.75,Z 576.503,A -85,B 0,C 180,E1 5172.3,E2 5172.3} C_VEL
LIN {X 0,Y 405.018,Z 584.149,A -85,B 0,C 180,E1 5169.623,E2 5169.623} C_VEL
LIN {X 0,Y 413.441,Z 590.602,A -85,B 0,C 180,E1 5167.281,E2 5167.281} C_VEL
LIN {X 0,Y 420.229,Z 595.799,A -85,B 0,C 180,E1 5165.3,E2 5165.3} C_VEL
LIN {X 0,Y 428.387,Z 601.723,A -85,B 0,C 180,E1 5162.831,E2 5162.831} C_VEL
LIN {X 0,Y 436.334,Z 607.697,A -85,B 0,C 180,E1 5160.24,E2 5160.24} C_VEL
LIN {X 0,Y 445.139,Z 613.695,A -85,B 0,C 180,E1 5157.188,E2 5157.188} C_VEL
LIN {X 0,Y 452.244,Z 619.182,A -85,B 0,C 180,E1 5154.368,E2 5154.368} C_VEL
LIN {X 0,Y 458.611,Z 623.134,A -85,B 0,C 180,E1 5151.752,E2 5151.752} C_VEL
LIN {X 0,Y 464.442,Z 627.782,A -85,B 0,C 180,E1 5148.838,E2 5148.838} C_VEL
LIN {X 0,Y 469.572,Z 631.192,A -85,B 0,C 180,E1 5146.068,E2 5146.068} C_VEL
LIN {X 0,Y 473.698,Z 633.36,A -85,B 0,C 180,E1 5143.549,E2 5143.549} C_VEL
LIN {X 0,Y 475.746,Z 634.747,A -85,B 0,C 180,E1 5142.008,E2 5142.008} C_VEL
LIN {X 0,Y 478.592,Z 637.36,A -85,B 0,C 180,E1 5139.256,E2 5139.256} C_VEL
LIN {X 0,Y 480.766,Z 639.092,A -85,B 0,C 180,E1 5136.567,E2 5136.567} C_VEL
LIN {X 0,Y 482.099,Z 640.052,A -85,B 0,C 180,E1 5134.162,E2 5134.162} C_VEL
LIN {X 0,Y 482.947,Z 640.557,A -85,B 0,C 180,E1 5131.661,E2 5131.661} C_VEL
LIN {X 0,Y 483.038,Z 640.594,A -85,B 0,C 180,E1 5129.288,E2 5129.288} C_VEL
LIN {X 0,Y 482.483,Z 640.276,A -85,B 0,C 180,E1 5126.674,E2 5126.674} C_VEL
LIN {X 0,Y 481.194,Z 639.383,A -85,B 0,C 180,E1 5124.037,E2 5124.037} C_VEL
LIN {X 0,Y 479.124,Z 637.842,A -85,B 0,C 180,E1 5121.359,E2 5121.359} C_VEL
LIN {X 0,Y 476.58,Z 635.562,A -85,B 0,C 180,E1 5118.75,E2 5118.75} C_VEL
LIN {X 0,Y 474.269,Z 633.623,A -85,B 0,C 180,E1 5116.841,E2 5116.841} C_VEL
LIN {X 0,Y 470.015,Z 631.449,A -85,B 0,C 180,E1 5114.201,E2 5114.201} C_VEL
LIN {X 0,Y 464.998,Z 628.188,A -85,B 0,C 180,E1 5111.446,E2 5111.446} C_VEL
LIN {X 0,Y 459.473,Z 623.751,A -85,B 0,C 180,E1 5108.655,E2 5108.655} C_VEL
LIN {X 0,Y 453.151,Z 619.8,A -85,B 0,C 180,E1 5105.994,E2 5105.994} C_VEL
LIN {X 0,Y 446.02,Z 614.434,A -85,B 0,C 180,E1 5103.156,E2 5103.156} C_VEL
LIN {X 0,Y 439.05,Z 609.666,A -85,B 0,C 180,E1 5100.721,E2 5100.721} C_VEL
LIN {X 0,Y 433.037,Z 605.203,A -85,B 0,C 180,E1 5098.687,E2 5098.687} C_VEL
LIN {X 0,Y 427.855,Z 601.372,A -85,B 0,C 180,E1 5097.013,E2 5097.013} C_VEL
LIN {X 0,Y 420.152,Z 595.736,A -85,B 0,C 180,E1 5094.675,E2 5094.675} C_VEL
LIN {X 0,Y 412.958,Z 590.256,A -85,B 0,C 180,E1 5092.578,E2 5092.578} C_VEL
LIN {X 0,Y 402.495,Z 582.258,A -85,B 0,C 180,E1 5089.699,E2 5089.699} C_VEL
LIN {X 0,Y 393.165,Z 575.258,A -85,B 0,C 180,E1 5087.306,E2 5087.306} C_VEL
LIN {X 0,Y 384.067,Z 568.41,A -85,B 0,C 180,E1 5085.083,E2 5085.083} C_VEL
LIN {X 0,Y 373.47,Z 560.303,A -85,B 0,C 180,E1 5082.638,E2 5082.638} C_VEL
LIN {X 0,Y 348.787,Z 539.862,A -85,B 0,C 180,E1 5076.196,E2 5076.196} C_VEL
LIN {X 0,Y 330.385,Z 520.551,A -85,B 0,C 180,E1 5070.008,E2 5070.008} C_VEL
LIN {X 0,Y 320.31,Z 506.996,A -85,B 0,C 180,E1 5065.765,E2 5065.765} C_VEL
LIN {X 0,Y 310.714,Z 489.893,A -85,B 0,C 180,E1 5060.633,E2 5060.633} C_VEL
LIN {X 0,Y 303.881,Z 470.608,A -85,B 0,C 180,E1 5055.213,E2 5055.213} C_VEL
LIN {X 0,Y 301.788,Z 462.981,A -85,B 0,C 180,E1 5052.874,E2 5052.874} C_VEL
LIN {X 0,Y 299.952,Z 456.715,A -85,B 0,C 180,E1 5050.419,E2 5050.419} C_VEL
LIN {X 0,Y 298.302,Z 451.583,A -85,B 0,C 180,E1 5047.608,E2 5047.608} C_VEL
LIN {X 0,Y 297.098,Z 447.621,A -85,B 0,C 180,E1 5044.439,E2 5044.439} C_VEL
LIN {X 0,Y 296.515,Z 445.614,A -85,B 0,C 180,E1 5040,E2 5040} C_VEL
LIN {X 0,Y 297.178,Z 447.974,A -85,B 0,C 180,E1 5035.562,E2 5035.562} C_VEL
LIN {X 0,Y 297.977,Z 450.647,A -85,B 0,C 180,E1 5033.378,E2 5033.378} C_VEL
LIN {X 0,Y 290.092,Z 516.419,A -85,B 0,C 180,E1 5032.515,E2 5032.515} C_VEL
LIN {X 0,Y 285.335,Z 540.566,A -85,B 0,C 180,E1 5032.132,E2 5032.132} C_VEL
LIN {X 0,Y 279.828,Z 560.183,A -85,B 0,C 180,E1 5031.748,E2 5031.748} C_VEL
LIN {X 0,Y 274.062,Z 576.794,A -85,B 0,C 180,E1 5031.334,E2 5031.334} C_VEL
LIN {X 0,Y 267.364,Z 593.038,A -85,B 0,C 180,E1 5030.813,E2 5030.813} C_VEL
LIN {X 0,Y 259.747,Z 608.894,A -85,B 0,C 180,E1 5030.174,E2 5030.174} C_VEL
LIN {X 0,Y 251.22,Z 624.328,A -85,B 0,C 180,E1 5029.407,E2 5029.407} C_VEL
LIN {X 0,Y 241.807,Z 639.3,A -85,B 0,C 180,E1 5028.486,E2 5028.486} C_VEL
LIN {X 0,Y 230.616,Z 655.021,A -85,B 0,C 180,E1 5027.267,E2 5027.267} C_VEL
LIN {X 0,Y 215.428,Z 673.473,A -85,B 0,C 180,E1 5025.375,E2 5025.375} C_VEL
LIN {X 0,Y 203.214,Z 686.464,A -85,B 0,C 180,E1 5023.606,E2 5023.606} C_VEL
LIN {X 0,Y 190.786,Z 698.345,A -85,B 0,C 180,E1 5021.527,E2 5021.527} C_VEL
LIN {X 0,Y 178.653,Z 708.834,A -85,B 0,C 180,E1 5019.154,E2 5019.154} C_VEL
LIN {X 0,Y 165.862,Z 718.865,A -85,B 0,C 180,E1 5016.177,E2 5016.177} C_VEL
LIN {X 0,Y 153.172,Z 727.901,A -85,B 0,C 180,E1 5012.582,E2 5012.582} C_VEL
LIN {X 0,Y 138.84,Z 737.22,A -85,B 0,C 180,E1 5007.404,E2 5007.404} C_VEL
LIN {X 0,Y 123.963,Z 745.875,A -85,B 0,C 180,E1 5000.011,E2 5000.011} C_VEL
LIN {X 0,Y 113.61,Z 751.5,A -85,B 0,C 180,E1 4992.655,E2 4992.655} C_VEL
LIN {X 0,Y 105.751,Z 755.685,A -85,B 0,C 180,E1 4984.557,E2 4984.557} C_VEL
LIN {X 0,Y 100.102,Z 758.808,A -85,B 0,C 180,E1 4975.433,E2 4975.433} C_VEL
LIN {X 0,Y 96.892,Z 760.899,A -85,B 0,C 180,E1 4965.561,E2 4965.561} C_VEL
LIN {X 0,Y 95.976,Z 761.939,A -85,B 0,C 180,E1 4955.979,E2 4955.979} C_VEL
LIN {X 0,Y 96.009,Z 762.182,A -85,B 0,C 180,E1 4948.807,E2 4948.807} C_VEL
LIN {X 0,Y 96.271,Z 761.531,A -85,B 0,C 180,E1 4938.62,E2 4938.62} C_VEL
LIN {X 0,Y 99.124,Z 759.408,A -85,B 0,C 180,E1 4926.837,E2 4926.837} C_VEL
LIN {X 0,Y 104.582,Z 756.315,A -85,B 0,C 180,E1 4916.983,E2 4916.983} C_VEL
LIN {X 0,Y 112.076,Z 752.314,A -85,B 0,C 180,E1 4908.692,E2 4908.692} C_VEL
LIN {X 0,Y 121.504,Z 747.213,A -85,B 0,C 180,E1 4901.517,E2 4901.517} C_VEL
LIN {X 0,Y 132.497,Z 740.956,A -85,B 0,C 180,E1 4895.421,E2 4895.421} C_VEL
LIN {X 0,Y 144.768,Z 733.445,A -85,B 0,C 180,E1 4890.279,E2 4890.279} C_VEL
LIN {X 0,Y 160.344,Z 723.024,A -85,B 0,C 180,E1 4885.3,E2 4885.3} C_VEL
LIN {X 0,Y 173.066,Z 713.456,A -85,B 0,C 180,E1 4882.084,E2 4882.084} C_VEL
LIN {X 0,Y 177.816,Z 709.254,A -85,B 0,C 180,E1 4880.642,E2 4880.642} C_VEL
LIN {X 0,Y 188.394,Z 698.519,A -85,B 0,C 180,E1 4876.465,E2 4876.465} C_VEL
LIN {X 0,Y 193.333,Z 693.806,A -85,B 0,C 180,E1 4875.333,E2 4875.333} C_VEL
LIN {X 0,Y 208.431,Z 678.786,A -85,B 0,C 180,E1 4873.169,E2 4873.169} C_VEL
LIN {X 0,Y 220.518,Z 665.252,A -85,B 0,C 180,E1 4871.687,E2 4871.687} C_VEL
LIN {X 0,Y 231.327,Z 651.696,A -85,B 0,C 180,E1 4870.513,E2 4870.513} C_VEL
LIN {X 0,Y 241.276,Z 637.702,A -85,B 0,C 180,E1 4869.537,E2 4869.537} C_VEL
LIN {X 0,Y 250.416,Z 623.221,A -85,B 0,C 180,E1 4868.727,E2 4868.727} C_VEL
LIN {X 0,Y 258.975,Z 607.798,A -85,B 0,C 180,E1 4868.029,E2 4868.029} C_VEL
LIN {X 0,Y 266.682,Z 591.801,A -85,B 0,C 180,E1 4867.444,E2 4867.444} C_VEL
LIN {X 0,Y 274.615,Z 572.393,A -85,B 0,C 180,E1 4866.89,E2 4866.89} C_VEL
LIN {X 0,Y 281.886,Z 549.651,A -85,B 0,C 180,E1 4866.42,E2 4866.42} C_VEL
LIN {X 0,Y 286.377,Z 531.191,A -85,B 0,C 180,E1 4866.125,E2 4866.125} C_VEL
LIN {X 0,Y 289.538,Z 513.465,A -85,B 0,C 180,E1 4865.873,E2 4865.873} C_VEL
LIN {X 0,Y 296.386,Z 456.945,A -85,B 0,C 180,E1 4865.139,E2 4865.139} C_VEL
LIN {X 0,Y 295.925,Z 455.271,A -85,B 0,C 180,E1 4863.487,E2 4863.487} C_VEL
LIN {X 0,Y 295.532,Z 453.63,A -85,B 0,C 180,E1 4859.612,E2 4859.612} C_VEL
LIN {X 0,Y 296.122,Z 455.899,A -85,B 0,C 180,E1 4855.449,E2 4855.449} C_VEL
LIN {X 0,Y 297.201,Z 459.572,A -85,B 0,C 180,E1 4852.558,E2 4852.558} C_VEL
LIN {X 0,Y 298.817,Z 465.005,A -85,B 0,C 180,E1 4849.687,E2 4849.687} C_VEL
LIN {X 0,Y 300.894,Z 472.784,A -85,B 0,C 180,E1 4846.842,E2 4846.842} C_VEL
LIN {X 0,Y 308.342,Z 496.316,A -85,B 0,C 180,E1 4840.142,E2 4840.142} C_VEL
LIN {X 0,Y 317.832,Z 514.13,A -85,B 0,C 180,E1 4834.719,E2 4834.719} C_VEL
LIN {X 0,Y 328.92,Z 529.481,A -85,B 0,C 180,E1 4829.794,E2 4829.794} C_VEL
LIN {X 0,Y 347.175,Z 548.69,A -85,B 0,C 180,E1 4823.45,E2 4823.45} C_VEL
LIN {X 0,Y 371.81,Z 568.918,A -85,B 0,C 180,E1 4816.916,E2 4816.916} C_VEL
LIN {X 0,Y 383.426,Z 577.829,A -85,B 0,C 180,E1 4814.181,E2 4814.181} C_VEL
LIN {X 0,Y 393.471,Z 585.52,A -85,B 0,C 180,E1 4811.659,E2 4811.659} C_VEL
LIN {X 0,Y 403.242,Z 592.838,A -85,B 0,C 180,E1 4809.093,E2 4809.093} C_VEL
LIN {X 0,Y 413.172,Z 600.224,A -85,B 0,C 180,E1 4806.305,E2 4806.305} C_VEL
LIN {X 0,Y 420.849,Z 606.18,A -85,B 0,C 180,E1 4803.985,E2 4803.985} C_VEL
LIN {X 0,Y 427.585,Z 610.916,A -85,B 0,C 180,E1 4801.899,E2 4801.899} C_VEL
LIN {X 0,Y 434.221,Z 615.973,A -85,B 0,C 180,E1 4799.671,E2 4799.671} C_VEL
LIN {X 0,Y 441.775,Z 621.104,A -85,B 0,C 180,E1 4797.057,E2 4797.057} C_VEL
LIN {X 0,Y 448.733,Z 626.407,A -85,B 0,C 180,E1 4794.306,E2 4794.306} C_VEL
LIN {X 0,Y 454.781,Z 630.154,A -85,B 0,C 180,E1 4791.809,E2 4791.809} C_VEL
LIN {X 0,Y 460.465,Z 634.666,A -85,B 0,C 180,E1 4789.007,E2 4789.007} C_VEL
LIN {X 0,Y 465.186,Z 637.878,A -85,B 0,C 180,E1 4786.48,E2 4786.48} C_VEL
LIN {X 0,Y 469.659,Z 640.294,A -85,B 0,C 180,E1 4783.793,E2 4783.793} C_VEL
LIN {X 0,Y 471.854,Z 641.628,A -85,B 0,C 180,E1 4782.232,E2 4782.232} C_VEL
LIN {X 0,Y 474.78,Z 644.326,A -85,B 0,C 180,E1 4779.453,E2 4779.453} C_VEL
LIN {X 0,Y 476.94,Z 646.079,A -85,B 0,C 180,E1 4776.862,E2 4776.862} C_VEL
LIN {X 0,Y 478.431,Z 647.143,A -85,B 0,C 180,E1 4774.314,E2 4774.314} C_VEL
LIN {X 0,Y 479.325,Z 647.687,A -85,B 0,C 180,E1 4771.793,E2 4771.793} C_VEL
LIN {X 0,Y 479.421,Z 647.73,A -85,B 0,C 180,E1 4769.283,E2 4769.283} C_VEL
LIN {X 0,Y 478.869,Z 647.413,A -85,B 0,C 180,E1 4766.649,E2 4766.649} C_VEL
LIN {X 0,Y 477.573,Z 646.511,A -85,B 0,C 180,E1 4763.992,E2 4763.992} C_VEL
LIN {X 0,Y 475.442,Z 644.925,A -85,B 0,C 180,E1 4761.283,E2 4761.283} C_VEL
LIN {X 0,Y 472.709,Z 642.476,A -85,B 0,C 180,E1 4758.533,E2 4758.533} C_VEL
LIN {X 0,Y 470.463,Z 640.672,A -85,B 0,C 180,E1 4756.732,E2 4756.732} C_VEL
LIN {X 0,Y 465.995,Z 638.359,A -85,B 0,C 180,E1 4754.004,E2 4754.004} C_VEL
LIN {X 0,Y 461.28,Z 635.271,A -85,B 0,C 180,E1 4751.422,E2 4751.422} C_VEL
LIN {X 0,Y 455.987,Z 631.043,A -85,B 0,C 180,E1 4748.74,E2 4748.74} C_VEL
LIN {X 0,Y 449.832,Z 627.149,A -85,B 0,C 180,E1 4746.14,E2 4746.14} C_VEL
LIN {X 0,Y 442.681,Z 621.852,A -85,B 0,C 180,E1 4743.293,E2 4743.293} C_VEL
LIN {X 0,Y 437.65,Z 618.305,A -85,B 0,C 180,E1 4741.482,E2 4741.482} C_VEL
LIN {X 0,Y 429.469,Z 612.429,A -85,B 0,C 180,E1 4738.727,E2 4738.727} C_VEL
LIN {X 0,Y 423.275,Z 607.882,A -85,B 0,C 180,E1 4736.746,E2 4736.746} C_VEL
LIN {X 0,Y 415.558,Z 602.171,A -85,B 0,C 180,E1 4734.417,E2 4734.417} C_VEL
LIN {X 0,Y 409.704,Z 597.697,A -85,B 0,C 180,E1 4732.713,E2 4732.713} C_VEL
LIN {X 0,Y 401.211,Z 591.231,A -85,B 0,C 180,E1 4730.362,E2 4730.362} C_VEL
LIN {X 0,Y 391.346,Z 583.896,A -85,B 0,C 180,E1 4727.788,E2 4727.788} C_VEL
LIN {X 0,Y 381.258,Z 576.226,A -85,B 0,C 180,E1 4725.294,E2 4725.294} C_VEL
LIN {X 0,Y 366.319,Z 564.77,A -85,B 0,C 180,E1 4721.76,E2 4721.76} C_VEL
LIN {X 0,Y 343.047,Z 544.702,A -85,B 0,C 180,E1 4715.248,E2 4715.248} C_VEL
LIN {X 0,Y 326.331,Z 526.198,A -85,B 0,C 180,E1 4709.156,E2 4709.156} C_VEL
LIN {X 0,Y 317.166,Z 513.021,A -85,B 0,C 180,E1 4704.939,E2 4704.939} C_VEL
LIN {X 0,Y 307.946,Z 495.395,A -85,B 0,C 180,E1 4699.588,E2 4699.588} C_VEL
LIN {X 0,Y 301.636,Z 475.821,A -85,B 0,C 180,E1 4694.053,E2 4694.053} C_VEL
LIN {X 0,Y 299.659,Z 468.103,A -85,B 0,C 180,E1 4691.549,E2 4691.549} C_VEL
LIN {X 0,Y 298.054,Z 462.413,A -85,B 0,C 180,E1 4689.072,E2 4689.072} C_VEL
LIN {X 0,Y 296.746,Z 457.995,A -85,B 0,C 180,E1 4686.384,E2 4686.384} C_VEL
LIN {X 0,Y 295.947,Z 455.312,A -85,B 0,C 180,E1 4683.874,E2 4683.874} C_VEL
LIN {X 0,Y 295.536,Z 453.581,A -85,B 0,C 180,E1 4680,E2 4680} C_VEL
LIN {X 0,Y 296.129,Z 455.901,A -85,B 0,C 180,E1 4675.74,E2 4675.74} C_VEL
LIN {X 0,Y 296.364,Z 457.241,A -85,B 0,C 180,E1 4674.831,E2 4674.831} C_VEL
LIN {X 0,Y 289.105,Z 516.593,A -85,B 0,C 180,E1 4674.086,E2 4674.086} C_VEL
LIN {X 0,Y 284.105,Z 541.304,A -85,B 0,C 180,E1 4673.718,E2 4673.718} C_VEL
LIN {X 0,Y 278.79,Z 560.007,A -85,B 0,C 180,E1 4673.38,E2 4673.38} C_VEL
LIN {X 0,Y 272.707,Z 577.286,A -85,B 0,C 180,E1 4672.983,E2 4672.983} C_VEL
LIN {X 0,Y 265.716,Z 593.924,A -85,B 0,C 180,E1 4672.486,E2 4672.486} C_VEL
LIN {X 0,Y 258.066,Z 609.538,A -85,B 0,C 180,E1 4671.899,E2 4671.899} C_VEL
LIN {X 0,Y 249.385,Z 624.958,A -85,B 0,C 180,E1 4671.184,E2 4671.184} C_VEL
LIN {X 0,Y 238.901,Z 641.255,A -85,B 0,C 180,E1 4670.237,E2 4670.237} C_VEL
LIN {X 0,Y 224.267,Z 660.772,A -85,B 0,C 180,E1 4668.734,E2 4668.734} C_VEL
LIN {X 0,Y 212.131,Z 674.793,A -85,B 0,C 180,E1 4667.309,E2 4667.309} C_VEL
LIN {X 0,Y 200.156,Z 687.176,A -85,B 0,C 180,E1 4665.697,E2 4665.697} C_VEL
LIN {X 0,Y 188.366,Z 698.167,A -85,B 0,C 180,E1 4663.875,E2 4663.875} C_VEL
LIN {X 0,Y 175.919,Z 708.656,A -85,B 0,C 180,E1 4661.635,E2 4661.635} C_VEL
LIN {X 0,Y 162.935,Z 718.543,A -85,B 0,C 180,E1 4658.853,E2 4658.853} C_VEL
LIN {X 0,Y 149.586,Z 727.723,A -85,B 0,C 180,E1 4655.36,E2 4655.36} C_VEL
LIN {X 0,Y 134.611,Z 737.041,A -85,B 0,C 180,E1 4650.337,E2 4650.337} C_VEL
LIN {X 0,Y 118.872,Z 745.696,A -85,B 0,C 180,E1 4643.033,E2 4643.033} C_VEL
LIN {X 0,Y 107.742,Z 751.321,A -85,B 0,C 180,E1 4635.602,E2 4635.602} C_VEL
LIN {X 0,Y 99.003,Z 755.57,A -85,B 0,C 180,E1 4627.072,E2 4627.072} C_VEL
LIN {X 0,Y 92.527,Z 758.781,A -85,B 0,C 180,E1 4616.988,E2 4616.988} C_VEL
LIN {X 0,Y 88.982,Z 760.813,A -85,B 0,C 180,E1 4606.313,E2 4606.313} C_VEL
LIN {X 0,Y 87.988,Z 761.763,A -85,B 0,C 180,E1 4596.524,E2 4596.524} C_VEL
LIN {X 0,Y 88.007,Z 762.007,A -85,B 0,C 180,E1 4588.698,E2 4588.698} C_VEL
LIN {X 0,Y 88.365,Z 761.355,A -85,B 0,C 180,E1 4577.586,E2 4577.586} C_VEL
LIN {X 0,Y 91.723,Z 759.22,A -85,B 0,C 180,E1 4564.797,E2 4564.797} C_VEL
LIN {X 0,Y 97.843,Z 756.137,A -85,B 0,C 180,E1 4554.379,E2 4554.379} C_VEL
LIN {X 0,Y 106.136,Z 752.105,A -85,B 0,C 180,E1 4545.725,E2 4545.725} C_VEL
LIN {X 0,Y 116.244,Z 747.034,A -85,B 0,C 180,E1 4538.497,E2 4538.497} C_VEL
LIN {X 0,Y 127.93,Z 740.777,A -85,B 0,C 180,E1 4532.434,E2 4532.434} C_VEL
LIN {X 0,Y 140.784,Z 733.29,A -85,B 0,C 180,E1 4527.418,E2 4527.418} C_VEL
LIN {X 0,Y 157.028,Z 722.845,A -85,B 0,C 180,E1 4522.605,E2 4522.605} C_VEL
LIN {X 0,Y 173.689,Z 710.44,A -85,B 0,C 180,E1 4518.807,E2 4518.807} C_VEL
LIN {X 0,Y 186.571,Z 699.749,A -85,B 0,C 180,E1 4516.427,E2 4516.427} C_VEL
LIN {X 0,Y 193.333,Z 693.806,A -85,B 0,C 180,E1 4515.333,E2 4515.333} C_VEL
LIN {X 0,Y 198.221,Z 688.993,A -85,B 0,C 180,E1 4514.273,E2 4514.273} C_VEL
LIN {X 0,Y 208.941,Z 676.505,A -85,B 0,C 180,E1 4511.008,E2 4511.008} C_VEL
LIN {X 0,Y 213.725,Z 671.208,A -85,B 0,C 180,E1 4510.178,E2 4510.178} C_VEL
LIN {X 0,Y 228.075,Z 654.037,A -85,B 0,C 180,E1 4508.711,E2 4508.711} C_VEL
LIN {X 0,Y 239.108,Z 638.947,A -85,B 0,C 180,E1 4507.718,E2 4507.718} C_VEL
LIN {X 0,Y 248.761,Z 623.976,A -85,B 0,C 180,E1 4506.939,E2 4506.939} C_VEL
LIN {X 0,Y 257.488,Z 608.542,A -85,B 0,C 180,E1 4506.293,E2 4506.293} C_VEL
LIN {X 0,Y 265.273,Z 592.686,A -85,B 0,C 180,E1 4505.757,E2 4505.757} C_VEL
LIN {X 0,Y 272.105,Z 576.443,A -85,B 0,C 180,E1 4505.32,E2 4505.32} C_VEL
LIN {X 0,Y 278.573,Z 558.031,A -85,B 0,C 180,E1 4504.942,E2 4504.942} C_VEL
LIN {X 0,Y 285.083,Z 533.669,A -85,B 0,C 180,E1 4504.562,E2 4504.562} C_VEL
LIN {X 0,Y 288.65,Z 514.492,A -85,B 0,C 180,E1 4504.305,E2 4504.305} C_VEL
LIN {X 0,Y 295,Z 463.349,A -85,B 0,C 180,E1 4503.692,E2 4503.692} C_VEL
LIN {X 0,Y 294.553,Z 461.602,A -85,B 0,C 180,E1 4499.611,E2 4499.611} C_VEL
LIN {X 0,Y 295.055,Z 463.708,A -85,B 0,C 180,E1 4495.724,E2 4495.724} C_VEL
LIN {X 0,Y 296.06,Z 467.41,A -85,B 0,C 180,E1 4492.822,E2 4492.822} C_VEL
LIN {X 0,Y 297.467,Z 472.607,A -85,B 0,C 180,E1 4490.129,E2 4490.129} C_VEL
LIN {X 0,Y 299.408,Z 480.578,A -85,B 0,C 180,E1 4487.267,E2 4487.267} C_VEL
LIN {X 0,Y 305.653,Z 501.814,A -85,B 0,C 180,E1 4481.202,E2 4481.202} C_VEL
LIN {X 0,Y 314.179,Z 519.454,A -85,B 0,C 180,E1 4475.761,E2 4475.761} C_VEL
LIN {X 0,Y 323.085,Z 532.968,A -85,B 0,C 180,E1 4471.334,E2 4471.334} C_VEL
LIN {X 0,Y 337.908,Z 550.074,A -85,B 0,C 180,E1 4465.534,E2 4465.534} C_VEL
LIN {X 0,Y 357.106,Z 567.418,A -85,B 0,C 180,E1 4459.699,E2 4459.699} C_VEL
LIN {X 0,Y 376.037,Z 582.268,A -85,B 0,C 180,E1 4454.984,E2 4454.984} C_VEL
LIN {X 0,Y 385.239,Z 589.203,A -85,B 0,C 180,E1 4452.732,E2 4452.732} C_VEL
LIN {X 0,Y 394.158,Z 595.869,A -85,B 0,C 180,E1 4450.444,E2 4450.444} C_VEL
LIN {X 0,Y 403.451,Z 603.002,A -85,B 0,C 180,E1 4447.919,E2 4447.919} C_VEL
LIN {X 0,Y 411.709,Z 609.237,A -85,B 0,C 180,E1 4445.551,E2 4445.551} C_VEL
LIN {X 0,Y 420.913,Z 615.907,A -85,B 0,C 180,E1 4442.761,E2 4442.761} C_VEL
LIN {X 0,Y 428.496,Z 621.659,A -85,B 0,C 180,E1 4440.263,E2 4440.263} C_VEL
LIN {X 0,Y 436.014,Z 626.714,A -85,B 0,C 180,E1 4437.724,E2 4437.724} C_VEL
LIN {X 0,Y 443.689,Z 632.611,A -85,B 0,C 180,E1 4434.742,E2 4434.742} C_VEL
LIN {X 0,Y 450.088,Z 636.69,A -85,B 0,C 180,E1 4432.122,E2 4432.122} C_VEL
LIN {X 0,Y 454.92,Z 640.403,A -85,B 0,C 180,E1 4429.826,E2 4429.826} C_VEL
LIN {X 0,Y 459.9,Z 643.999,A -85,B 0,C 180,E1 4427.196,E2 4427.196} C_VEL
LIN {X 0,Y 464.677,Z 646.734,A -85,B 0,C 180,E1 4424.452,E2 4424.452} C_VEL
LIN {X 0,Y 467.812,Z 648.474,A -85,B 0,C 180,E1 4422.37,E2 4422.37} C_VEL
LIN {X 0,Y 470.685,Z 651.132,A -85,B 0,C 180,E1 4419.66,E2 4419.66} C_VEL
LIN {X 0,Y 472.937,Z 653,A -85,B 0,C 180,E1 4416.921,E2 4416.921} C_VEL
LIN {X 0,Y 474.422,Z 654.063,A -85,B 0,C 180,E1 4414.351,E2 4414.351} C_VEL
LIN {X 0,Y 475.331,Z 654.619,A -85,B 0,C 180,E1 4411.808,E2 4411.808} C_VEL
LIN {X 0,Y 475.44,Z 654.667,A -85,B 0,C 180,E1 4409.398,E2 4409.398} C_VEL
LIN {X 0,Y 474.945,Z 654.381,A -85,B 0,C 180,E1 4406.863,E2 4406.863} C_VEL
LIN {X 0,Y 473.686,Z 653.517,A -85,B 0,C 180,E1 4404.186,E2 4404.186} C_VEL
LIN {X 0,Y 471.699,Z 652.048,A -85,B 0,C 180,E1 4401.468,E2 4401.468} C_VEL
LIN {X 0,Y 469.147,Z 649.776,A -85,B 0,C 180,E1 4398.818,E2 4398.818} C_VEL
LIN {X 0,Y 466.821,Z 647.778,A -85,B 0,C 180,E1 4396.879,E2 4396.879} C_VEL
LIN {X 0,Y 462.381,Z 645.507,A -85,B 0,C 180,E1 4394.191,E2 4394.191} C_VEL
LIN {X 0,Y 457.288,Z 642.197,A -85,B 0,C 180,E1 4391.386,E2 4391.386} C_VEL
LIN {X 0,Y 451.706,Z 637.734,A -85,B 0,C 180,E1 4388.581,E2 4388.581} C_VEL
LIN {X 0,Y 445.056,Z 633.557,A -85,B 0,C 180,E1 4385.804,E2 4385.804} C_VEL
LIN {X 0,Y 437.838,Z 628.099,A -85,B 0,C 180,E1 4382.955,E2 4382.955} C_VEL
LIN {X 0,Y 430.785,Z 623.304,A -85,B 0,C 180,E1 4380.507,E2 4380.507} C_VEL
LIN {X 0,Y 423.283,Z 617.626,A -85,B 0,C 180,E1 4377.999,E2 4377.999} C_VEL
LIN {X 0,Y 416.034,Z 612.529,A -85,B 0,C 180,E1 4375.768,E2 4375.768} C_VEL
LIN {X 0,Y 407.817,Z 606.103,A -85,B 0,C 180,E1 4373.297,E2 4373.297} C_VEL
LIN {X 0,Y 397.761,Z 598.634,A -85,B 0,C 180,E1 4370.51,E2 4370.51} C_VEL
LIN {X 0,Y 388.391,Z 591.664,A -85,B 0,C 180,E1 4368.075,E2 4368.075} C_VEL
LIN {X 0,Y 379.858,Z 585.096,A -85,B 0,C 180,E1 4365.94,E2 4365.94} C_VEL
LIN {X 0,Y 367.202,Z 575.408,A -85,B 0,C 180,E1 4362.902,E2 4362.902} C_VEL
LIN {X 0,Y 344.2,Z 556.32,A -85,B 0,C 180,E1 4356.55,E2 4356.55} C_VEL
LIN {X 0,Y 325.903,Z 536.72,A -85,B 0,C 180,E1 4349.905,E2 4349.905} C_VEL
LIN {X 0,Y 315.273,Z 521.369,A -85,B 0,C 180,E1 4344.849,E2 4344.849} C_VEL
LIN {X 0,Y 307.126,Z 505.449,A -85,B 0,C 180,E1 4339.89,E2 4339.89} C_VEL
LIN {X 0,Y 300.697,Z 486.265,A -85,B 0,C 180,E1 4334.343,E2 4334.343} C_VEL
LIN {X 0,Y 298.742,Z 477.811,A -85,B 0,C 180,E1 4331.83,E2 4331.83} C_VEL
LIN {X 0,Y 297.157,Z 471.439,A -85,B 0,C 180,E1 4329.344,E2 4329.344} C_VEL
LIN {X 0,Y 295.816,Z 466.527,A -85,B 0,C 180,E1 4326.599,E2 4326.599} C_VEL
LIN {X 0,Y 294.918,Z 463.193,A -85,B 0,C 180,E1 4323.693,E2 4323.693} C_VEL
LIN {X 0,Y 294.558,Z 461.551,A -85,B 0,C 180,E1 4320,E2 4320} C_VEL
LIN {X 0,Y 294.978,Z 463.545,A -85,B 0,C 180,E1 4316.302,E2 4316.302} C_VEL
LIN {X 0,Y 288.331,Z 516.803,A -85,B 0,C 180,E1 4315.666,E2 4315.666} C_VEL
LIN {X 0,Y 283.115,Z 541.965,A -85,B 0,C 180,E1 4315.318,E2 4315.318} C_VEL
LIN {X 0,Y 277.734,Z 560.575,A -85,B 0,C 180,E1 4315.009,E2 4315.009} C_VEL
LIN {X 0,Y 271.761,Z 577.319,A -85,B 0,C 180,E1 4314.658,E2 4314.658} C_VEL
LIN {X 0,Y 264.785,Z 593.748,A -85,B 0,C 180,E1 4314.211,E2 4314.211} C_VEL
LIN {X 0,Y 257.146,Z 609.19,A -85,B 0,C 180,E1 4313.683,E2 4313.683} C_VEL
LIN {X 0,Y 248.277,Z 624.781,A -85,B 0,C 180,E1 4313.023,E2 4313.023} C_VEL
LIN {X 0,Y 237.665,Z 641.078,A -85,B 0,C 180,E1 4312.157,E2 4312.157} C_VEL
LIN {X 0,Y 222.827,Z 660.595,A -85,B 0,C 180,E1 4310.776,E2 4310.776} C_VEL
LIN {X 0,Y 210.498,Z 674.616,A -85,B 0,C 180,E1 4309.463,E2 4309.463} C_VEL
LIN {X 0,Y 198.306,Z 686.999,A -85,B 0,C 180,E1 4307.971,E2 4307.971} C_VEL
LIN {X 0,Y 186.271,Z 697.989,A -85,B 0,C 180,E1 4306.279,E2 4306.279} C_VEL
LIN {X 0,Y 173.524,Z 708.478,A -85,B 0,C 180,E1 4304.188,E2 4304.188} C_VEL
LIN {X 0,Y 160.172,Z 718.365,A -85,B 0,C 180,E1 4301.576,E2 4301.576} C_VEL
LIN {X 0,Y 146.369,Z 727.544,A -85,B 0,C 180,E1 4298.268,E2 4298.268} C_VEL
LIN {X 0,Y 130.757,Z 736.863,A -85,B 0,C 180,E1 4293.452,E2 4293.452} C_VEL
LIN {X 0,Y 114.14,Z 745.517,A -85,B 0,C 180,E1 4286.315,E2 4286.315} C_VEL
LIN {X 0,Y 102.189,Z 751.142,A -85,B 0,C 180,E1 4278.879,E2 4278.879} C_VEL
LIN {X 0,Y 92.77,Z 755.328,A -85,B 0,C 180,E1 4270.286,E2 4270.286} C_VEL
LIN {X 0,Y 85.686,Z 758.453,A -85,B 0,C 180,E1 4260.113,E2 4260.113} C_VEL
LIN {X 0,Y 81.401,Z 760.545,A -85,B 0,C 180,E1 4248.622,E2 4248.622} C_VEL
LIN {X 0,Y 80.002,Z 761.587,A -85,B 0,C 180,E1 4237.179,E2 4237.179} C_VEL
LIN {X 0,Y 80.004,Z 761.832,A -85,B 0,C 180,E1 4228.568,E2 4228.568} C_VEL
LIN {X 0,Y 80.49,Z 761.178,A -85,B 0,C 180,E1 4216.35,E2 4216.35} C_VEL
LIN {X 0,Y 84.414,Z 759.052,A -85,B 0,C 180,E1 4202.491,E2 4202.491} C_VEL
LIN {X 0,Y 91.335,Z 755.958,A -85,B 0,C 180,E1 4191.397,E2 4191.397} C_VEL
LIN {X 0,Y 100.379,Z 751.957,A -85,B 0,C 180,E1 4182.521,E2 4182.521} C_VEL
LIN {X 0,Y 111.336,Z 746.856,A -85,B 0,C 180,E1 4175.2,E2 4175.2} C_VEL
LIN {X 0,Y 123.736,Z 740.599,A -85,B 0,C 180,E1 4169.237,E2 4169.237} C_VEL
LIN {X 0,Y 137.212,Z 733.111,A -85,B 0,C 180,E1 4164.387,E2 4164.387} C_VEL
LIN {X 0,Y 154.074,Z 722.667,A -85,B 0,C 180,E1 4159.801,E2 4159.801} C_VEL
LIN {X 0,Y 170.826,Z 710.582,A -85,B 0,C 180,E1 4156.301,E2 4156.301} C_VEL
LIN {X 0,Y 184.435,Z 699.571,A -85,B 0,C 180,E1 4154.001,E2 4154.001} C_VEL
LIN {X 0,Y 197.374,Z 687.888,A -85,B 0,C 180,E1 4152.151,E2 4152.151} C_VEL
LIN {X 0,Y 210.027,Z 675.114,A -85,B 0,C 180,E1 4150.591,E2 4150.591} C_VEL
LIN {X 0,Y 213.725,Z 671.208,A -85,B 0,C 180,E1 4150.178,E2 4150.178} C_VEL
LIN {X 0,Y 218.446,Z 665.789,A -85,B 0,C 180,E1 4149.399,E2 4149.399} C_VEL
LIN {X 0,Y 228.749,Z 651.767,A -85,B 0,C 180,E1 4146.805,E2 4146.805} C_VEL
LIN {X 0,Y 233.143,Z 645.875,A -85,B 0,C 180,E1 4146.188,E2 4146.188} C_VEL
LIN {X 0,Y 246.451,Z 626.215,A -85,B 0,C 180,E1 4145.192,E2 4145.192} C_VEL
LIN {X 0,Y 255.75,Z 610.206,A -85,B 0,C 180,E1 4144.569,E2 4144.569} C_VEL
LIN {X 0,Y 263.604,Z 594.634,A -85,B 0,C 180,E1 4144.082,E2 4144.082} C_VEL
LIN {X 0,Y 270.493,Z 578.753,A -85,B 0,C 180,E1 4143.687,E2 4143.687} C_VEL
LIN {X 0,Y 276.411,Z 562.627,A -85,B 0,C 180,E1 4143.375,E2 4143.375} C_VEL
LIN {X 0,Y 281.595,Z 545.413,A -85,B 0,C 180,E1 4143.111,E2 4143.111} C_VEL
LIN {X 0,Y 285.759,Z 527.745,A -85,B 0,C 180,E1 4142.879,E2 4142.879} C_VEL
LIN {X 0,Y 289.112,Z 507.939,A -85,B 0,C 180,E1 4142.64,E2 4142.64} C_VEL
LIN {X 0,Y 293.694,Z 470.609,A -85,B 0,C 180,E1 4142.207,E2 4142.207} C_VEL
LIN {X 0,Y 293.574,Z 469.573,A -85,B 0,C 180,E1 4139.61,E2 4139.61} C_VEL
LIN {X 0,Y 294.014,Z 471.632,A -85,B 0,C 180,E1 4135.905,E2 4135.905} C_VEL
LIN {X 0,Y 294.925,Z 475.247,A -85,B 0,C 180,E1 4133.087,E2 4133.087} C_VEL
LIN {X 0,Y 296.215,Z 480.546,A -85,B 0,C 180,E1 4130.43,E2 4130.43} C_VEL
LIN {X 0,Y 297.898,Z 488.269,A -85,B 0,C 180,E1 4127.743,E2 4127.743} C_VEL
LIN {X 0,Y 302.993,Z 507.427,A -85,B 0,C 180,E1 4122.227,E2 4122.227} C_VEL
LIN {X 0,Y 310.231,Z 524.242,A -85,B 0,C 180,E1 4116.996,E2 4116.996} C_VEL
LIN {X 0,Y 318.748,Z 538.367,A -85,B 0,C 180,E1 4112.286,E2 4112.286} C_VEL
LIN {X 0,Y 332.956,Z 555.744,A -85,B 0,C 180,E1 4106.25,E2 4106.25} C_VEL
LIN {X 0,Y 352.56,Z 573.914,A -85,B 0,C 180,E1 4099.925,E2 4099.925} C_VEL
LIN {X 0,Y 372.857,Z 589.866,A -85,B 0,C 180,E1 4094.712,E2 4094.712} C_VEL
LIN {X 0,Y 382.638,Z 597.295,A -85,B 0,C 180,E1 4092.309,E2 4092.309} C_VEL
LIN {X 0,Y 393.09,Z 605.098,A -85,B 0,C 180,E1 4089.58,E2 4089.58} C_VEL
LIN {X 0,Y 401.617,Z 611.529,A -85,B 0,C 180,E1 4087.222,E2 4087.222} C_VEL
LIN {X 0,Y 409.584,Z 617.675,A -85,B 0,C 180,E1 4084.889,E2 4084.889} C_VEL
LIN {X 0,Y 417.905,Z 623.5,A -85,B 0,C 180,E1 4082.371,E2 4082.371} C_VEL
LIN {X 0,Y 426.591,Z 630.117,A -85,B 0,C 180,E1 4079.482,E2 4079.482} C_VEL
LIN {X 0,Y 433.474,Z 634.8,A -85,B 0,C 180,E1 4077.078,E2 4077.078} C_VEL
LIN {X 0,Y 440.708,Z 640.265,A -85,B 0,C 180,E1 4074.243,E2 4074.243} C_VEL
LIN {X 0,Y 447.649,Z 644.683,A -85,B 0,C 180,E1 4071.341,E2 4071.341} C_VEL
LIN {X 0,Y 452.927,Z 648.895,A -85,B 0,C 180,E1 4068.667,E2 4068.667} C_VEL
LIN {X 0,Y 458.23,Z 652.344,A -85,B 0,C 180,E1 4065.783,E2 4065.783} C_VEL
LIN {X 0,Y 462.451,Z 654.517,A -85,B 0,C 180,E1 4063.247,E2 4063.247} C_VEL
LIN {X 0,Y 464.926,Z 656.578,A -85,B 0,C 180,E1 4061.159,E2 4061.159} C_VEL
LIN {X 0,Y 467.463,Z 658.846,A -85,B 0,C 180,E1 4058.486,E2 4058.486} C_VEL
LIN {X 0,Y 469.496,Z 660.338,A -85,B 0,C 180,E1 4055.744,E2 4055.744} C_VEL
LIN {X 0,Y 470.797,Z 661.209,A -85,B 0,C 180,E1 4052.921,E2 4052.921} C_VEL
LIN {X 0,Y 471.333,Z 661.502,A -85,B 0,C 180,E1 4050.365,E2 4050.365} C_VEL
LIN {X 0,Y 470.996,Z 661.316,A -85,B 0,C 180,E1 4047.567,E2 4047.567} C_VEL
LIN {X 0,Y 469.884,Z 660.601,A -85,B 0,C 180,E1 4044.873,E2 4044.873} C_VEL
LIN {X 0,Y 468.089,Z 659.343,A -85,B 0,C 180,E1 4042.267,E2 4042.267} C_VEL
LIN {X 0,Y 465.601,Z 657.17,A -85,B 0,C 180,E1 4039.484,E2 4039.484} C_VEL
LIN {X 0,Y 462.806,Z 654.67,A -85,B 0,C 180,E1 4037.004,E2 4037.004} C_VEL
LIN {X 0,Y 458.612,Z 652.552,A -85,B 0,C 180,E1 4034.447,E2 4034.447} C_VEL
LIN {X 0,Y 453.501,Z 649.309,A -85,B 0,C 180,E1 4031.624,E2 4031.624} C_VEL
LIN {X 0,Y 448.265,Z 645.211,A -85,B 0,C 180,E1 4028.957,E2 4028.957} C_VEL
LIN {X 0,Y 443.918,Z 642.333,A -85,B 0,C 180,E1 4027.069,E2 4027.069} C_VEL
LIN {X 0,Y 437.548,Z 638.02,A -85,B 0,C 180,E1 4024.51,E2 4024.51} C_VEL
LIN {X 0,Y 431.165,Z 633.128,A -85,B 0,C 180,E1 4022.071,E2 4022.071} C_VEL
LIN {X 0,Y 423.076,Z 627.577,A -85,B 0,C 180,E1 4019.347,E2 4019.347} C_VEL
LIN {X 0,Y 415.951,Z 622.215,A -85,B 0,C 180,E1 4017.03,E2 4017.03} C_VEL
LIN {X 0,Y 406.502,Z 615.276,A -85,B 0,C 180,E1 4014.173,E2 4014.173} C_VEL
LIN {X 0,Y 397.15,Z 608.27,A -85,B 0,C 180,E1 4011.536,E2 4011.536} C_VEL
LIN {X 0,Y 388.948,Z 601.984,A -85,B 0,C 180,E1 4009.321,E2 4009.321} C_VEL
LIN {X 0,Y 379.407,Z 594.75,A -85,B 0,C 180,E1 4006.887,E2 4006.887} C_VEL
LIN {X 0,Y 368.428,Z 586.475,A -85,B 0,C 180,E1 4004.226,E2 4004.226} C_VEL
LIN {X 0,Y 343.794,Z 566.284,A -85,B 0,C 180,E1 3997.435,E2 3997.435} C_VEL
LIN {X 0,Y 326.509,Z 548.443,A -85,B 0,C 180,E1 3991.219,E2 3991.219} C_VEL
LIN {X 0,Y 314.142,Z 531.306,A -85,B 0,C 180,E1 3985.302,E2 3985.302} C_VEL
LIN {X 0,Y 305.585,Z 514.065,A -85,B 0,C 180,E1 3979.795,E2 3979.795} C_VEL
LIN {X 0,Y 299.225,Z 494.554,A -85,B 0,C 180,E1 3974.02,E2 3974.02} C_VEL
LIN {X 0,Y 297.193,Z 484.957,A -85,B 0,C 180,E1 3971.204,E2 3971.204} C_VEL
LIN {X 0,Y 295.774,Z 478.7,A -85,B 0,C 180,E1 3968.75,E2 3968.75} C_VEL
LIN {X 0,Y 294.591,Z 473.922,A -85,B 0,C 180,E1 3966.04,E2 3966.04} C_VEL
LIN {X 0,Y 293.847,Z 470.978,A -85,B 0,C 180,E1 3963.316,E2 3963.316} C_VEL
LIN {X 0,Y 293.579,Z 469.523,A -85,B 0,C 180,E1 3960,E2 3960} C_VEL
LIN {X 0,Y 293.68,Z 470.751,A -85,B 0,C 180,E1 3957.776,E2 3957.776} C_VEL
LIN {X 0,Y 287.759,Z 517.132,A -85,B 0,C 180,E1 3957.252,E2 3957.252} C_VEL
LIN {X 0,Y 282.54,Z 541.915,A -85,B 0,C 180,E1 3956.937,E2 3956.937} C_VEL
LIN {X 0,Y 277.152,Z 560.399,A -85,B 0,C 180,E1 3956.662,E2 3956.662} C_VEL
LIN {X 0,Y 271.478,Z 576.268,A -85,B 0,C 180,E1 3956.368,E2 3956.368} C_VEL
LIN {X 0,Y 264.587,Z 592.511,A -85,B 0,C 180,E1 3955.976,E2 3955.976} C_VEL
LIN {X 0,Y 256.73,Z 608.366,A -85,B 0,C 180,E1 3955.494,E2 3955.494} C_VEL
LIN {X 0,Y 247.869,Z 623.877,A -85,B 0,C 180,E1 3954.908,E2 3954.908} C_VEL
LIN {X 0,Y 238.158,Z 638.771,A -85,B 0,C 180,E1 3954.207,E2 3954.207} C_VEL
LIN {X 0,Y 226.507,Z 654.491,A -85,B 0,C 180,E1 3953.265,E2 3953.265} C_VEL
LIN {X 0,Y 210.912,Z 672.622,A -85,B 0,C 180,E1 3951.823,E2 3951.823} C_VEL
LIN {X 0,Y 197.687,Z 685.966,A -85,B 0,C 180,E1 3950.391,E2 3950.391} C_VEL
LIN {X 0,Y 184.511,Z 697.812,A -85,B 0,C 180,E1 3948.733,E2 3948.733} C_VEL
LIN {X 0,Y 171.484,Z 708.3,A -85,B 0,C 180,E1 3946.807,E2 3946.807} C_VEL
LIN {X 0,Y 157.784,Z 718.187,A -85,B 0,C 180,E1 3944.387,E2 3944.387} C_VEL
LIN {X 0,Y 143.668,Z 727.29,A -85,B 0,C 180,E1 3941.328,E2 3941.328} C_VEL
LIN {X 0,Y 128.145,Z 736.215,A -85,B 0,C 180,E1 3937.015,E2 3937.015} C_VEL
LIN {X 0,Y 109.814,Z 745.339,A -85,B 0,C 180,E1 3929.869,E2 3929.869} C_VEL
LIN {X 0,Y 97.007,Z 750.964,A -85,B 0,C 180,E1 3922.519,E2 3922.519} C_VEL
LIN {X 0,Y 86.703,Z 755.15,A -85,B 0,C 180,E1 3913.776,E2 3913.776} C_VEL
LIN {X 0,Y 78.719,Z 758.286,A -85,B 0,C 180,E1 3903.035,E2 3903.035} C_VEL
LIN {X 0,Y 73.764,Z 760.368,A -85,B 0,C 180,E1 3890.633,E2 3890.633} C_VEL
LIN {X 0,Y 72.025,Z 761.411,A -85,B 0,C 180,E1 3877.979,E2 3877.979} C_VEL
LIN {X 0,Y 72.001,Z 761.657,A -85,B 0,C 180,E1 3868.409,E2 3868.409} C_VEL
LIN {X 0,Y 72.658,Z 761.002,A -85,B 0,C 180,E1 3854.845,E2 3854.845} C_VEL
LIN {X 0,Y 77.289,Z 758.875,A -85,B 0,C 180,E1 3839.704,E2 3839.704} C_VEL
LIN {X 0,Y 85.11,Z 755.78,A -85,B 0,C 180,E1 3827.967,E2 3827.967} C_VEL
LIN {X 0,Y 95.046,Z 751.778,A -85,B 0,C 180,E1 3818.888,E2 3818.888} C_VEL
LIN {X 0,Y 106.843,Z 746.671,A -85,B 0,C 180,E1 3811.606,E2 3811.606} C_VEL
LIN {X 0,Y 119.954,Z 740.42,A -85,B 0,C 180,E1 3805.826,E2 3805.826} C_VEL
LIN {X 0,Y 134.044,Z 732.932,A -85,B 0,C 180,E1 3801.204,E2 3801.204} C_VEL
LIN {X 0,Y 151.633,Z 722.406,A -85,B 0,C 180,E1 3796.867,E2 3796.867} C_VEL
LIN {X 0,Y 168.72,Z 710.404,A -85,B 0,C 180,E1 3793.643,E2 3793.643} C_VEL
LIN {X 0,Y 182.637,Z 699.393,A -85,B 0,C 180,E1 3791.524,E2 3791.524} C_VEL
LIN {X 0,Y 195.825,Z 687.71,A -85,B 0,C 180,E1 3789.826,E2 3789.826} C_VEL
LIN {X 0,Y 208.21,Z 675.436,A -85,B 0,C 180,E1 3788.451,E2 3788.451} C_VEL
LIN {X 0,Y 219.962,Z 662.403,A -85,B 0,C 180,E1 3787.313,E2 3787.313} C_VEL
LIN {X 0,Y 232.325,Z 646.935,A -85,B 0,C 180,E1 3786.253,E2 3786.253} C_VEL
LIN {X 0,Y 233.143,Z 645.875,A -85,B 0,C 180,E1 3786.188,E2 3786.188} C_VEL
LIN {X 0,Y 237.45,Z 639.872,A -85,B 0,C 180,E1 3785.605,E2 3785.605} C_VEL
LIN {X 0,Y 247.402,Z 623.603,A -85,B 0,C 180,E1 3783.4,E2 3783.4} C_VEL
LIN {X 0,Y 250.732,Z 618.075,A -85,B 0,C 180,E1 3783.026,E2 3783.026} C_VEL
LIN {X 0,Y 262.163,Z 596.581,A -85,B 0,C 180,E1 3782.388,E2 3782.388} C_VEL
LIN {X 0,Y 269.599,Z 579.821,A -85,B 0,C 180,E1 3782.011,E2 3782.011} C_VEL
LIN {X 0,Y 275.744,Z 563.382,A -85,B 0,C 180,E1 3781.727,E2 3781.727} C_VEL
LIN {X 0,Y 281.057,Z 546.038,A -85,B 0,C 180,E1 3781.489,E2 3781.489} C_VEL
LIN {X 0,Y 285.251,Z 528.601,A -85,B 0,C 180,E1 3781.283,E2 3781.283} C_VEL
LIN {X 0,Y 288.429,Z 510.575,A -85,B 0,C 180,E1 3781.081,E2 3781.081} C_VEL
LIN {X 0,Y 292.59,Z 477.825,A -85,B 0,C 180,E1 3780.685,E2 3780.685} C_VEL
LIN {X 0,Y 292.596,Z 477.545,A -85,B 0,C 180,E1 3779.608,E2 3779.608} C_VEL
LIN {X 0,Y 292.959,Z 479.439,A -85,B 0,C 180,E1 3776.184,E2 3776.184} C_VEL
LIN {X 0,Y 293.758,Z 482.939,A -85,B 0,C 180,E1 3773.453,E2 3773.453} C_VEL
LIN {X 0,Y 294.894,Z 488.156,A -85,B 0,C 180,E1 3770.879,E2 3770.879} C_VEL
LIN {X 0,Y 296.312,Z 495.522,A -85,B 0,C 180,E1 3768.368,E2 3768.368} C_VEL
LIN {X 0,Y 300.666,Z 513.815,A -85,B 0,C 180,E1 3763.033,E2 3763.033} C_VEL
LIN {X 0,Y 307.579,Z 531.43,A -85,B 0,C 180,E1 3757.443,E2 3757.443} C_VEL
LIN {X 0,Y 315.731,Z 545.673,A -85,B 0,C 180,E1 3752.562,E2 3752.562} C_VEL
LIN {X 0,Y 328.87,Z 562.333,A -85,B 0,C 180,E1 3746.612,E2 3746.612} C_VEL
LIN {X 0,Y 347.957,Z 580.374,A -85,B 0,C 180,E1 3740.147,E2 3740.147} C_VEL
LIN {X 0,Y 366.194,Z 594.857,A -85,B 0,C 180,E1 3735.213,E2 3735.213} C_VEL
LIN {X 0,Y 377.161,Z 603.164,A -85,B 0,C 180,E1 3732.523,E2 3732.523} C_VEL
LIN {X 0,Y 387.23,Z 610.634,A -85,B 0,C 180,E1 3729.923,E2 3729.923} C_VEL
LIN {X 0,Y 395.413,Z 616.93,A -85,B 0,C 180,E1 3727.675,E2 3727.675} C_VEL
LIN {X 0,Y 401.929,Z 621.851,A -85,B 0,C 180,E1 3725.806,E2 3725.806} C_VEL
LIN {X 0,Y 409.814,Z 627.717,A -85,B 0,C 180,E1 3723.443,E2 3723.443} C_VEL
LIN {X 0,Y 415.642,Z 631.933,A -85,B 0,C 180,E1 3721.613,E2 3721.613} C_VEL
LIN {X 0,Y 423.773,Z 637.877,A -85,B 0,C 180,E1 3718.91,E2 3718.91} C_VEL
LIN {X 0,Y 429.581,Z 641.924,A -85,B 0,C 180,E1 3716.839,E2 3716.839} C_VEL
LIN {X 0,Y 435.825,Z 646.619,A -85,B 0,C 180,E1 3714.381,E2 3714.381} C_VEL
LIN {X 0,Y 442.959,Z 651.134,A -85,B 0,C 180,E1 3711.447,E2 3711.447} C_VEL
LIN {X 0,Y 448.594,Z 655.63,A -85,B 0,C 180,E1 3708.584,E2 3708.584} C_VEL
LIN {X 0,Y 453.65,Z 658.92,A -85,B 0,C 180,E1 3705.859,E2 3705.859} C_VEL
LIN {X 0,Y 458.139,Z 661.22,A -85,B 0,C 180,E1 3703.118,E2 3703.118} C_VEL
LIN {X 0,Y 461.048,Z 663.73,A -85,B 0,C 180,E1 3700.621,E2 3700.621} C_VEL
LIN {X 0,Y 463.497,Z 665.878,A -85,B 0,C 180,E1 3697.935,E2 3697.935} C_VEL
LIN {X 0,Y 465.375,Z 667.207,A -85,B 0,C 180,E1 3695.3,E2 3695.3} C_VEL
LIN {X 0,Y 466.438,Z 667.906,A -85,B 0,C 180,E1 3692.703,E2 3692.703} C_VEL
LIN {X 0,Y 466.877,Z 668.146,A -85,B 0,C 180,E1 3690,E2 3690} C_VEL
LIN {X 0,Y 466.504,Z 667.935,A -85,B 0,C 180,E1 3687.298,E2 3687.298} C_VEL
LIN {X 0,Y 465.277,Z 667.137,A -85,B 0,C 180,E1 3684.575,E2 3684.575} C_VEL
LIN {X 0,Y 463.259,Z 665.695,A -85,B 0,C 180,E1 3681.811,E2 3681.811} C_VEL
LIN {X 0,Y 460.759,Z 663.484,A -85,B 0,C 180,E1 3679.119,E2 3679.119} C_VEL
LIN {X 0,Y 458.118,Z 661.207,A -85,B 0,C 180,E1 3676.882,E2 3676.882} C_VEL
LIN {X 0,Y 453.628,Z 658.907,A -85,B 0,C 180,E1 3674.14,E2 3674.14} C_VEL
LIN {X 0,Y 448.487,Z 655.554,A -85,B 0,C 180,E1 3671.357,E2 3671.357} C_VEL
LIN {X 0,Y 442.817,Z 651.012,A -85,B 0,C 180,E1 3668.483,E2 3668.483} C_VEL
LIN {X 0,Y 435.37,Z 646.308,A -85,B 0,C 180,E1 3665.433,E2 3665.433} C_VEL
LIN {X 0,Y 428.618,Z 641.131,A -85,B 0,C 180,E1 3662.795,E2 3662.795} C_VEL
LIN {X 0,Y 421.305,Z 636.186,A -85,B 0,C 180,E1 3660.267,E2 3660.267} C_VEL
LIN {X 0,Y 412.295,Z 629.388,A -85,B 0,C 180,E1 3657.303,E2 3657.303} C_VEL
LIN {X 0,Y 403.905,Z 623.398,A -85,B 0,C 180,E1 3654.779,E2 3654.779} C_VEL
LIN {X 0,Y 396.442,Z 617.671,A -85,B 0,C 180,E1 3652.607,E2 3652.607} C_VEL
LIN {X 0,Y 386.755,Z 610.249,A -85,B 0,C 180,E1 3649.93,E2 3649.93} C_VEL
LIN {X 0,Y 375.247,Z 601.657,A -85,B 0,C 180,E1 3646.996,E2 3646.996} C_VEL
LIN {X 0,Y 358.736,Z 588.988,A -85,B 0,C 180,E1 3642.851,E2 3642.851} C_VEL
LIN {X 0,Y 337.037,Z 570.708,A -85,B 0,C 180,E1 3636.395,E2 3636.395} C_VEL
LIN {X 0,Y 319.658,Z 551.306,A -85,B 0,C 180,E1 3629.413,E2 3629.413} C_VEL
LIN {X 0,Y 309.535,Z 535.329,A -85,B 0,C 180,E1 3623.866,E2 3623.866} C_VEL
LIN {X 0,Y 302.089,Z 517.965,A -85,B 0,C 180,E1 3618.229,E2 3618.229} C_VEL
LIN {X 0,Y 297.011,Z 499.227,A -85,B 0,C 180,E1 3612.689,E2 3612.689} C_VEL
LIN {X 0,Y 295.535,Z 491.444,A -85,B 0,C 180,E1 3610.33,E2 3610.33} C_VEL
LIN {X 0,Y 294.379,Z 485.757,A -85,B 0,C 180,E1 3608.054,E2 3608.054} C_VEL
LIN {X 0,Y 293.364,Z 481.193,A -85,B 0,C 180,E1 3605.378,E2 3605.378} C_VEL
LIN {X 0,Y 292.827,Z 478.859,A -85,B 0,C 180,E1 3603.132,E2 3603.132} C_VEL
LIN {X 0,Y 292.6,Z 477.495,A -85,B 0,C 180,E1 3600,E2 3600} C_VEL
LIN {X 0,Y 292.562,Z 478.088,A -85,B 0,C 180,E1 3599.263,E2 3599.263} C_VEL
LIN {X 0,Y 287.303,Z 518.121,A -85,B 0,C 180,E1 3598.836,E2 3598.836} C_VEL
LIN {X 0,Y 282.138,Z 542.061,A -85,B 0,C 180,E1 3598.558,E2 3598.558} C_VEL
LIN {X 0,Y 276.8,Z 560.224,A -85,B 0,C 180,E1 3598.32,E2 3598.32} C_VEL
LIN {X 0,Y 271.088,Z 576.092,A -85,B 0,C 180,E1 3598.062,E2 3598.062} C_VEL
LIN {X 0,Y 264.144,Z 592.336,A -85,B 0,C 180,E1 3597.715,E2 3597.715} C_VEL
LIN {X 0,Y 256.223,Z 608.19,A -85,B 0,C 180,E1 3597.289,E2 3597.289} C_VEL
LIN {X 0,Y 247.331,Z 623.623,A -85,B 0,C 180,E1 3596.773,E2 3596.773} C_VEL
LIN {X 0,Y 237.318,Z 638.826,A -85,B 0,C 180,E1 3596.134,E2 3596.134} C_VEL
LIN {X 0,Y 224.723,Z 655.573,A -85,B 0,C 180,E1 3595.23,E2 3595.23} C_VEL
LIN {X 0,Y 209.116,Z 673.263,A -85,B 0,C 180,E1 3593.943,E2 3593.943} C_VEL
LIN {X 0,Y 195.567,Z 686.644,A -85,B 0,C 180,E1 3592.631,E2 3592.631} C_VEL
LIN {X 0,Y 182.745,Z 697.924,A -85,B 0,C 180,E1 3591.187,E2 3591.187} C_VEL
LIN {X 0,Y 168.868,Z 708.823,A -85,B 0,C 180,E1 3589.349,E2 3589.349} C_VEL
LIN {X 0,Y 154.861,Z 718.627,A -85,B 0,C 180,E1 3587.116,E2 3587.116} C_VEL
LIN {X 0,Y 139.336,Z 728.27,A -85,B 0,C 180,E1 3584.043,E2 3584.043} C_VEL
LIN {X 0,Y 119.163,Z 739.041,A -85,B 0,C 180,E1 3578.633,E2 3578.633} C_VEL
LIN {X 0,Y 104.354,Z 745.829,A -85,B 0,C 180,E1 3572.996,E2 3572.996} C_VEL
LIN {X 0,Y 91.548,Z 751.057,A -85,B 0,C 180,E1 3566.095,E2 3566.095} C_VEL
LIN {X 0,Y 80.406,Z 755.182,A -85,B 0,C 180,E1 3557.188,E2 3557.188} C_VEL
LIN {X 0,Y 71.624,Z 758.247,A -85,B 0,C 180,E1 3545.891,E2 3545.891} C_VEL
LIN {X 0,Y 66.004,Z 760.281,A -85,B 0,C 180,E1 3532.251,E2 3532.251} C_VEL
LIN {X 0,Y 64.026,Z 761.267,A -85,B 0,C 180,E1 3518.079,E2 3518.079} C_VEL
LIN {X 0,Y 63.997,Z 761.482,A -85,B 0,C 180,E1 3508.209,E2 3508.209} C_VEL
LIN {X 0,Y 65.038,Z 760.734,A -85,B 0,C 180,E1 3492.095,E2 3492.095} C_VEL
LIN {X 0,Y 70.785,Z 758.547,A -85,B 0,C 180,E1 3475.601,E2 3475.601} C_VEL
LIN {X 0,Y 79.817,Z 755.392,A -85,B 0,C 180,E1 3463.408,E2 3463.408} C_VEL
LIN {X 0,Y 90.839,Z 751.328,A -85,B 0,C 180,E1 3454.368,E2 3454.368} C_VEL
LIN {X 0,Y 103.565,Z 746.164,A -85,B 0,C 180,E1 3447.363,E2 3447.363} C_VEL
LIN {X 0,Y 117.468,Z 739.841,A -85,B 0,C 180,E1 3441.923,E2 3441.923} C_VEL
LIN {X 0,Y 133.968,Z 731.347,A -85,B 0,C 180,E1 3437.212,E2 3437.212} C_VEL
LIN {X 0,Y 153.014,Z 719.864,A -85,B 0,C 180,E1 3433.213,E2 3433.213} C_VEL
LIN {X 0,Y 167.927,Z 709.524,A -85,B 0,C 180,E1 3430.788,E2 3430.788} C_VEL
LIN {X 0,Y 181.188,Z 699.216,A -85,B 0,C 180,E1 3429.002,E2 3429.002} C_VEL
LIN {X 0,Y 194.604,Z 687.533,A -85,B 0,C 180,E1 3427.47,E2 3427.47} C_VEL
LIN {X 0,Y 207.173,Z 675.259,A -85,B 0,C 180,E1 3426.231,E2 3426.231} C_VEL
LIN {X 0,Y 219.345,Z 661.921,A -85,B 0,C 180,E1 3425.19,E2 3425.19} C_VEL
LIN {X 0,Y 232.654,Z 645.386,A -85,B 0,C 180,E1 3424.19,E2 3424.19} C_VEL
LIN {X 0,Y 245.852,Z 626.039,A -85,B 0,C 180,E1 3423.32,E2 3423.32} C_VEL
LIN {X 0,Y 250.732,Z 618.075,A -85,B 0,C 180,E1 3423.026,E2 3423.026} C_VEL
LIN {X 0,Y 254.478,Z 611.557,A -85,B 0,C 180,E1 3422.585,E2 3422.585} C_VEL
LIN {X 0,Y 262.649,Z 594.98,A -85,B 0,C 180,E1 3420.822,E2 3420.822} C_VEL
LIN {X 0,Y 265.847,Z 588.118,A -85,B 0,C 180,E1 3420.461,E2 3420.461} C_VEL
LIN {X 0,Y 274.682,Z 565.994,A -85,B 0,C 180,E1 3420.096,E2 3420.096} C_VEL
LIN {X 0,Y 280.614,Z 547.147,A -85,B 0,C 180,E1 3419.868,E2 3419.868} C_VEL
LIN {X 0,Y 284.996,Z 529.321,A -85,B 0,C 180,E1 3419.681,E2 3419.681} C_VEL
LIN {X 0,Y 288.203,Z 511.619,A -85,B 0,C 180,E1 3419.5,E2 3419.5} C_VEL
LIN {X 0,Y 291.609,Z 485.703,A -85,B 0,C 180,E1 3419.214,E2 3419.214} C_VEL
LIN {X 0,Y 291.926,Z 487.361,A -85,B 0,C 180,E1 3416.367,E2 3416.367} C_VEL
LIN {X 0,Y 292.601,Z 490.647,A -85,B 0,C 180,E1 3413.821,E2 3413.821} C_VEL
LIN {X 0,Y 293.587,Z 495.801,A -85,B 0,C 180,E1 3411.332,E2 3411.332} C_VEL
LIN {X 0,Y 294.735,Z 502.6,A -85,B 0,C 180,E1 3409.048,E2 3409.048} C_VEL
LIN {X 0,Y 298.718,Z 521.745,A -85,B 0,C 180,E1 3403.37,E2 3403.37} C_VEL
LIN {X 0,Y 304.87,Z 538.835,A -85,B 0,C 180,E1 3397.791,E2 3397.791} C_VEL
LIN {X 0,Y 312.4,Z 552.692,A -85,B 0,C 180,E1 3392.916,E2 3392.916} C_VEL
LIN {X 0,Y 325.896,Z 570.163,A -85,B 0,C 180,E1 3386.477,E2 3386.477} C_VEL
LIN {X 0,Y 344.198,Z 587.534,A -85,B 0,C 180,E1 3380.059,E2 3380.059} C_VEL
LIN {X 0,Y 365.273,Z 604.149,A -85,B 0,C 180,E1 3374.262,E2 3374.262} C_VEL
LIN {X 0,Y 375.274,Z 611.804,A -85,B 0,C 180,E1 3371.751,E2 3371.751} C_VEL
LIN {X 0,Y 385.377,Z 619.383,A -85,B 0,C 180,E1 3369.124,E2 3369.124} C_VEL
LIN {X 0,Y 395.089,Z 626.594,A -85,B 0,C 180,E1 3366.409,E2 3366.409} C_VEL
LIN {X 0,Y 402.662,Z 632.455,A -85,B 0,C 180,E1 3364.134,E2 3364.134} C_VEL
LIN {X 0,Y 409.739,Z 637.448,A -85,B 0,C 180,E1 3361.97,E2 3361.97} C_VEL
LIN {X 0,Y 417.62,Z 643.361,A -85,B 0,C 180,E1 3359.365,E2 3359.365} C_VEL
LIN {X 0,Y 424.305,Z 647.933,A -85,B 0,C 180,E1 3357.029,E2 3357.029} C_VEL
LIN {X 0,Y 430.729,Z 652.815,A -85,B 0,C 180,E1 3354.496,E2 3354.496} C_VEL
LIN {X 0,Y 437.32,Z 656.947,A -85,B 0,C 180,E1 3351.831,E2 3351.831} C_VEL
LIN {X 0,Y 443.117,Z 661.535,A -85,B 0,C 180,E1 3348.959,E2 3348.959} C_VEL
LIN {X 0,Y 447.76,Z 664.685,A -85,B 0,C 180,E1 3346.473,E2 3346.473} C_VEL
LIN {X 0,Y 452.658,Z 667.335,A -85,B 0,C 180,E1 3343.607,E2 3343.607} C_VEL
LIN {X 0,Y 454.791,Z 668.771,A -85,B 0,C 180,E1 3342.054,E2 3342.054} C_VEL
LIN {X 0,Y 457.512,Z 671.252,A -85,B 0,C 180,E1 3339.433,E2 3339.433} C_VEL
LIN {X 0,Y 459.75,Z 673.043,A -85,B 0,C 180,E1 3336.618,E2 3336.618} C_VEL
LIN {X 0,Y 461.128,Z 674.036,A -85,B 0,C 180,E1 3334.093,E2 3334.093} C_VEL
LIN {X 0,Y 461.934,Z 674.52,A -85,B 0,C 180,E1 3331.364,E2 3331.364} C_VEL
LIN {X 0,Y 462.01,Z 674.541,A -85,B 0,C 180,E1 3329.132,E2 3329.132} C_VEL
LIN {X 0,Y 461.445,Z 674.216,A -85,B 0,C 180,E1 3326.646,E2 3326.646} C_VEL
LIN {X 0,Y 460.152,Z 673.32,A -85,B 0,C 180,E1 3324.014,E2 3324.014} C_VEL
LIN {X 0,Y 458.165,Z 671.84,A -85,B 0,C 180,E1 3321.34,E2 3321.34} C_VEL
LIN {X 0,Y 455.679,Z 669.619,A -85,B 0,C 180,E1 3318.74,E2 3318.74} C_VEL
LIN {X 0,Y 453.389,Z 667.672,A -85,B 0,C 180,E1 3316.872,E2 3316.872} C_VEL
LIN {X 0,Y 448.502,Z 665.124,A -85,B 0,C 180,E1 3313.954,E2 3313.954} C_VEL
LIN {X 0,Y 443.951,Z 662.146,A -85,B 0,C 180,E1 3311.478,E2 3311.478} C_VEL
LIN {X 0,Y 438.237,Z 657.602,A -85,B 0,C 180,E1 3308.576,E2 3308.576} C_VEL
LIN {X 0,Y 432.132,Z 653.77,A -85,B 0,C 180,E1 3306.061,E2 3306.061} C_VEL
LIN {X 0,Y 425.179,Z 648.651,A -85,B 0,C 180,E1 3303.313,E2 3303.313} C_VEL
LIN {X 0,Y 420.025,Z 644.978,A -85,B 0,C 180,E1 3301.453,E2 3301.453} C_VEL
LIN {X 0,Y 411.768,Z 639.065,A -85,B 0,C 180,E1 3298.696,E2 3298.696} C_VEL
LIN {X 0,Y 406.01,Z 634.799,A -85,B 0,C 180,E1 3296.859,E2 3296.859} C_VEL
LIN {X 0,Y 397.441,Z 628.498,A -85,B 0,C 180,E1 3294.297,E2 3294.297} C_VEL
LIN {X 0,Y 391.441,Z 623.926,A -85,B 0,C 180,E1 3292.565,E2 3292.565} C_VEL
LIN {X 0,Y 382.751,Z 617.302,A -85,B 0,C 180,E1 3290.178,E2 3290.178} C_VEL
LIN {X 0,Y 373.123,Z 610.166,A -85,B 0,C 180,E1 3287.699,E2 3287.699} C_VEL
LIN {X 0,Y 361.683,Z 601.475,A -85,B 0,C 180,E1 3284.827,E2 3284.827} C_VEL
LIN {X 0,Y 340.786,Z 584.744,A -85,B 0,C 180,E1 3278.895,E2 3278.895} C_VEL
LIN {X 0,Y 322,Z 565.764,A -85,B 0,C 180,E1 3271.863,E2 3271.863} C_VEL
LIN {X 0,Y 308.937,Z 547.078,A -85,B 0,C 180,E1 3265.041,E2 3265.041} C_VEL
LIN {X 0,Y 301.438,Z 530.271,A -85,B 0,C 180,E1 3259.372,E2 3259.372} C_VEL
LIN {X 0,Y 296.807,Z 514.063,A -85,B 0,C 180,E1 3254.286,E2 3254.286} C_VEL
LIN {X 0,Y 294.098,Z 498.725,A -85,B 0,C 180,E1 3249.738,E2 3249.738} C_VEL
LIN {X 0,Y 293.066,Z 493.017,A -85,B 0,C 180,E1 3247.449,E2 3247.449} C_VEL
LIN {X 0,Y 292.218,Z 488.787,A -85,B 0,C 180,E1 3244.907,E2 3244.907} C_VEL
LIN {X 0,Y 291.775,Z 486.645,A -85,B 0,C 180,E1 3242.75,E2 3242.75} C_VEL
LIN {X 0,Y 291.594,Z 485.81,A -85,B 0,C 180,E1 3240.756,E2 3240.756} C_VEL
LIN {X 0,Y 286.861,Z 520.406,A -85,B 0,C 180,E1 3240.41,E2 3240.41} C_VEL
LIN {X 0,Y 281.775,Z 542.899,A -85,B 0,C 180,E1 3240.176,E2 3240.176} C_VEL
LIN {X 0,Y 276.431,Z 560.795,A -85,B 0,C 180,E1 3239.972,E2 3239.972} C_VEL
LIN {X 0,Y 270.436,Z 577.161,A -85,B 0,C 180,E1 3239.739,E2 3239.739} C_VEL
LIN {X 0,Y 263.447,Z 593.222,A -85,B 0,C 180,E1 3239.437,E2 3239.437} C_VEL
LIN {X 0,Y 255.471,Z 608.934,A -85,B 0,C 180,E1 3239.065,E2 3239.065} C_VEL
LIN {X 0,Y 246.014,Z 625.058,A -85,B 0,C 180,E1 3238.587,E2 3238.587} C_VEL
LIN {X 0,Y 233.106,Z 644.059,A -85,B 0,C 180,E1 3237.853,E2 3237.853} C_VEL
LIN {X 0,Y 219.255,Z 661.184,A -85,B 0,C 180,E1 3236.956,E2 3236.956} C_VEL
LIN {X 0,Y 206.706,Z 674.822,A -85,B 0,C 180,E1 3236.027,E2 3236.027} C_VEL
LIN {X 0,Y 193.715,Z 687.355,A -85,B 0,C 180,E1 3234.912,E2 3234.912} C_VEL
LIN {X 0,Y 180.094,Z 699.038,A -85,B 0,C 180,E1 3233.554,E2 3233.554} C_VEL
LIN {X 0,Y 164.677,Z 710.749,A -85,B 0,C 180,E1 3231.717,E2 3231.717} C_VEL
LIN {X 0,Y 144.77,Z 723.759,A -85,B 0,C 180,E1 3228.702,E2 3228.702} C_VEL
LIN {X 0,Y 129.034,Z 732.575,A -85,B 0,C 180,E1 3225.579,E2 3225.579} C_VEL
LIN {X 0,Y 113.785,Z 740.063,A -85,B 0,C 180,E1 3221.608,E2 3221.608} C_VEL
LIN {X 0,Y 99.238,Z 746.32,A -85,B 0,C 180,E1 3216.457,E2 3216.457} C_VEL
LIN {X 0,Y 85.73,Z 751.421,A -85,B 0,C 180,E1 3209.65,E2 3209.65} C_VEL
LIN {X 0,Y 73.159,Z 755.633,A -85,B 0,C 180,E1 3199.93,E2 3199.93} C_VEL
LIN {X 0,Y 61.612,Z 759.265,A -85,B 0,C 180,E1 3183.484,E2 3183.484} C_VEL
LIN {X 0,Y 56.24,Z 761.003,A -85,B 0,C 180,E1 3162.082,E2 3162.082} C_VEL
LIN {X 0,Y 56.008,Z 761.33,A -85,B 0,C 180,E1 3148.743,E2 3148.743} C_VEL
LIN {X 0,Y 57.195,Z 760.648,A -85,B 0,C 180,E1 3130.603,E2 3130.603} C_VEL
LIN {X 0,Y 63.764,Z 758.519,A -85,B 0,C 180,E1 3112.303,E2 3112.303} C_VEL
LIN {X 0,Y 73.797,Z 755.423,A -85,B 0,C 180,E1 3099.448,E2 3099.448} C_VEL
LIN {X 0,Y 85.73,Z 751.421,A -85,B 0,C 180,E1 3090.349,E2 3090.349} C_VEL
LIN {X 0,Y 99.238,Z 746.319,A -85,B 0,C 180,E1 3083.543,E2 3083.543} C_VEL
LIN {X 0,Y 113.785,Z 740.063,A -85,B 0,C 180,E1 3078.391,E2 3078.391} C_VEL
LIN {X 0,Y 129.035,Z 732.575,A -85,B 0,C 180,E1 3074.421,E2 3074.421} C_VEL
LIN {X 0,Y 147.588,Z 722.132,A -85,B 0,C 180,E1 3070.82,E2 3070.82} C_VEL
LIN {X 0,Y 165.636,Z 710.048,A -85,B 0,C 180,E1 3068.158,E2 3068.158} C_VEL
LIN {X 0,Y 180.094,Z 699.038,A -85,B 0,C 180,E1 3066.446,E2 3066.446} C_VEL
LIN {X 0,Y 193.716,Z 687.355,A -85,B 0,C 180,E1 3065.088,E2 3065.088} C_VEL
LIN {X 0,Y 206.703,Z 674.825,A -85,B 0,C 180,E1 3063.974,E2 3063.974} C_VEL
LIN {X 0,Y 219.255,Z 661.184,A -85,B 0,C 180,E1 3063.043,E2 3063.043} C_VEL
LIN {X 0,Y 233.602,Z 643.388,A -85,B 0,C 180,E1 3062.117,E2 3062.117} C_VEL
LIN {X 0,Y 246.014,Z 625.058,A -85,B 0,C 180,E1 3061.414,E2 3061.414} C_VEL
LIN {X 0,Y 255.471,Z 608.934,A -85,B 0,C 180,E1 3060.935,E2 3060.935} C_VEL
LIN {X 0,Y 263.448,Z 593.221,A -85,B 0,C 180,E1 3060.563,E2 3060.563} C_VEL
LIN {X 0,Y 265.847,Z 588.118,A -85,B 0,C 180,E1 3060.461,E2 3060.461} C_VEL
LIN {X 0,Y 268.92,Z 581.165,A -85,B 0,C 180,E1 3060.121,E2 3060.121} C_VEL
LIN {X 0,Y 275.535,Z 563.571,A -85,B 0,C 180,E1 3058.61,E2 3058.61} C_VEL
LIN {X 0,Y 277.991,Z 556.35,A -85,B 0,C 180,E1 3058.319,E2 3058.319} C_VEL
LIN {X 0,Y 284.398,Z 532.697,A -85,B 0,C 180,E1 3058.103,E2 3058.103} C_VEL
LIN {X 0,Y 288.044,Z 513.656,A -85,B 0,C 180,E1 3057.928,E2 3057.928} C_VEL
LIN {X 0,Y 290.721,Z 494.384,A -85,B 0,C 180,E1 3057.743,E2 3057.743} C_VEL
LIN {X 0,Y 290.945,Z 495.619,A -85,B 0,C 180,E1 3056.256,E2 3056.256} C_VEL
LIN {X 0,Y 291.488,Z 498.598,A -85,B 0,C 180,E1 3054.07,E2 3054.07} C_VEL
LIN {X 0,Y 292.279,Z 503.318,A -85,B 0,C 180,E1 3051.838,E2 3051.838} C_VEL
LIN {X 0,Y 293.041,Z 509.816,A -85,B 0,C 180,E1 3049.681,E2 3049.681} C_VEL
LIN {X 0,Y 295.359,Z 524.301,A -85,B 0,C 180,E1 3045.342,E2 3045.342} C_VEL
LIN {X 0,Y 299.695,Z 540.289,A -85,B 0,C 180,E1 3040.173,E2 3040.173} C_VEL
LIN {X 0,Y 307.135,Z 556.794,A -85,B 0,C 180,E1 3034.343,E2 3034.343} C_VEL
LIN {X 0,Y 318.865,Z 573.592,A -85,B 0,C 180,E1 3027.998,E2 3027.998} C_VEL
LIN {X 0,Y 336.495,Z 591.488,A -85,B 0,C 180,E1 3021.172,E2 3021.172} C_VEL
LIN {X 0,Y 355.942,Z 607.152,A -85,B 0,C 180,E1 3015.389,E2 3015.389} C_VEL
LIN {X 0,Y 368.416,Z 616.628,A -85,B 0,C 180,E1 3012.189,E2 3012.189} C_VEL
LIN {X 0,Y 379.166,Z 624.673,A -85,B 0,C 180,E1 3009.406,E2 3009.406} C_VEL
LIN {X 0,Y 389.029,Z 631.979,A -85,B 0,C 180,E1 3006.687,E2 3006.687} C_VEL
LIN {X 0,Y 396.495,Z 637.837,A -85,B 0,C 180,E1 3004.448,E2 3004.448} C_VEL
LIN {X 0,Y 403.538,Z 642.719,A -85,B 0,C 180,E1 3002.335,E2 3002.335} C_VEL
LIN {X 0,Y 411.514,Z 648.83,A -85,B 0,C 180,E1 2999.71,E2 2999.71} C_VEL
LIN {X 0,Y 419.05,Z 653.968,A -85,B 0,C 180,E1 2997.109,E2 2997.109} C_VEL
LIN {X 0,Y 426.922,Z 659.876,A -85,B 0,C 180,E1 2994.018,E2 2994.018} C_VEL
LIN {X 0,Y 433.287,Z 663.893,A -85,B 0,C 180,E1 2991.381,E2 2991.381} C_VEL
LIN {X 0,Y 438.833,Z 668.304,A -85,B 0,C 180,E1 2988.582,E2 2988.582} C_VEL
LIN {X 0,Y 444.295,Z 671.823,A -85,B 0,C 180,E1 2985.587,E2 2985.587} C_VEL
LIN {X 0,Y 448.855,Z 674.16,A -85,B 0,C 180,E1 2982.87,E2 2982.87} C_VEL
LIN {X 0,Y 451.876,Z 676.909,A -85,B 0,C 180,E1 2980.066,E2 2980.066} C_VEL
LIN {X 0,Y 454.185,Z 678.888,A -85,B 0,C 180,E1 2977.335,E2 2977.335} C_VEL
LIN {X 0,Y 455.805,Z 680.025,A -85,B 0,C 180,E1 2974.781,E2 2974.781} C_VEL
LIN {X 0,Y 456.812,Z 680.688,A -85,B 0,C 180,E1 2972.258,E2 2972.258} C_VEL
LIN {X 0,Y 457.067,Z 680.816,A -85,B 0,C 180,E1 2969.624,E2 2969.624} C_VEL
LIN {X 0,Y 456.653,Z 680.571,A -85,B 0,C 180,E1 2967.114,E2 2967.114} C_VEL
LIN {X 0,Y 455.426,Z 679.75,A -85,B 0,C 180,E1 2964.457,E2 2964.457} C_VEL
LIN {X 0,Y 453.465,Z 678.34,A -85,B 0,C 180,E1 2961.761,E2 2961.761} C_VEL
LIN {X 0,Y 450.933,Z 676.095,A -85,B 0,C 180,E1 2959.008,E2 2959.008} C_VEL
LIN {X 0,Y 448.432,Z 673.972,A -85,B 0,C 180,E1 2956.856,E2 2956.856} C_VEL
LIN {X 0,Y 443.629,Z 671.445,A -85,B 0,C 180,E1 2954.042,E2 2954.042} C_VEL
LIN {X 0,Y 438.232,Z 667.867,A -85,B 0,C 180,E1 2951.098,E2 2951.098} C_VEL
LIN {X 0,Y 432.614,Z 663.371,A -85,B 0,C 180,E1 2948.3,E2 2948.3} C_VEL
LIN {X 0,Y 425.929,Z 659.201,A -85,B 0,C 180,E1 2945.6,E2 2945.6} C_VEL
LIN {X 0,Y 418.565,Z 653.566,A -85,B 0,C 180,E1 2942.703,E2 2942.703} C_VEL
LIN {X 0,Y 410.224,Z 647.905,A -85,B 0,C 180,E1 2939.865,E2 2939.865} C_VEL
LIN {X 0,Y 401.571,Z 641.423,A -85,B 0,C 180,E1 2937.047,E2 2937.047} C_VEL
LIN {X 0,Y 392.023,Z 634.411,A -85,B 0,C 180,E1 2934.203,E2 2934.203} C_VEL
LIN {X 0,Y 384.348,Z 628.644,A -85,B 0,C 180,E1 2932.024,E2 2932.024} C_VEL
LIN {X 0,Y 375.456,Z 621.801,A -85,B 0,C 180,E1 2929.611,E2 2929.611} C_VEL
LIN {X 0,Y 365.692,Z 614.496,A -85,B 0,C 180,E1 2927.12,E2 2927.12} C_VEL
LIN {X 0,Y 345.664,Z 599.115,A -85,B 0,C 180,E1 2921.706,E2 2921.706} C_VEL
LIN {X 0,Y 324.344,Z 579.756,A -85,B 0,C 180,E1 2914.344,E2 2914.344} C_VEL
LIN {X 0,Y 310.078,Z 561.609,A -85,B 0,C 180,E1 2907.46,E2 2907.46} C_VEL
LIN {X 0,Y 302.808,Z 548.039,A -85,B 0,C 180,E1 2902.522,E2 2902.522} C_VEL
LIN {X 0,Y 297.03,Z 531.543,A -85,B 0,C 180,E1 2896.929,E2 2896.929} C_VEL
LIN {X 0,Y 293.592,Z 513.878,A -85,B 0,C 180,E1 2891.492,E2 2891.492} C_VEL
LIN {X 0,Y 292.534,Z 505.336,A -85,B 0,C 180,E1 2888.897,E2 2888.897} C_VEL
LIN {X 0,Y 291.753,Z 500.071,A -85,B 0,C 180,E1 2886.741,E2 2886.741} C_VEL
LIN {X 0,Y 291.068,Z 496.271,A -85,B 0,C 180,E1 2884.334,E2 2884.334} C_VEL
LIN {X 0,Y 290.765,Z 494.527,A -85,B 0,C 180,E1 2882.562,E2 2882.562} C_VEL
LIN {X 0,Y 290.703,Z 494.52,A -85,B 0,C 180,E1 2882.249,E2 2882.249} C_VEL
LIN {X 0,Y 286.368,Z 523.477,A -85,B 0,C 180,E1 2881.982,E2 2881.982} C_VEL
LIN {X 0,Y 281.663,Z 543.651,A -85,B 0,C 180,E1 2881.798,E2 2881.798} C_VEL
LIN {X 0,Y 276.293,Z 561.372,A -85,B 0,C 180,E1 2881.626,E2 2881.626} C_VEL
LIN {X 0,Y 270.016,Z 578.233,A -85,B 0,C 180,E1 2881.422,E2 2881.422} C_VEL
LIN {X 0,Y 262.488,Z 595.176,A -85,B 0,C 180,E1 2881.148,E2 2881.148} C_VEL
LIN {X 0,Y 251.957,Z 615.185,A -85,B 0,C 180,E1 2880.721,E2 2880.721} C_VEL
LIN {X 0,Y 239.942,Z 633.982,A -85,B 0,C 180,E1 2880.186,E2 2880.186} C_VEL
LIN {X 0,Y 228.948,Z 648.923,A -85,B 0,C 180,E1 2879.632,E2 2879.632} C_VEL
LIN {X 0,Y 217.48,Z 662.687,A -85,B 0,C 180,E1 2878.983,E2 2878.983} C_VEL
LIN {X 0,Y 205.548,Z 675.404,A -85,B 0,C 180,E1 2878.222,E2 2878.222} C_VEL
LIN {X 0,Y 193.165,Z 687.178,A -85,B 0,C 180,E1 2877.312,E2 2877.312} C_VEL
LIN {X 0,Y 179.363,Z 698.86,A -85,B 0,C 180,E1 2876.136,E2 2876.136} C_VEL
LIN {X 0,Y 164.677,Z 709.87,A -85,B 0,C 180,E1 2874.648,E2 2874.648} C_VEL
LIN {X 0,Y 146.276,Z 721.954,A -85,B 0,C 180,E1 2872.321,E2 2872.321} C_VEL
LIN {X 0,Y 127.092,Z 732.473,A -85,B 0,C 180,E1 2869.116,E2 2869.116} C_VEL
LIN {X 0,Y 111.475,Z 739.884,A -85,B 0,C 180,E1 2865.6,E2 2865.6} C_VEL
LIN {X 0,Y 96.263,Z 746.141,A -85,B 0,C 180,E1 2860.925,E2 2860.925} C_VEL
LIN {X 0,Y 81.904,Z 751.242,A -85,B 0,C 180,E1 2854.592,E2 2854.592} C_VEL
LIN {X 0,Y 67.957,Z 755.525,A -85,B 0,C 180,E1 2844.982,E2 2844.982} C_VEL
LIN {X 0,Y 54.546,Z 759.199,A -85,B 0,C 180,E1 2827.218,E2 2827.218} C_VEL
LIN {X 0,Y 48.404,Z 760.819,A -85,B 0,C 180,E1 2804.35,E2 2804.35} C_VEL
LIN {X 0,Y 48.007,Z 761.161,A -85,B 0,C 180,E1 2788.746,E2 2788.746} C_VEL
LIN {X 0,Y 49.632,Z 760.471,A -85,B 0,C 180,E1 2767.497,E2 2767.497} C_VEL
LIN {X 0,Y 57.535,Z 758.341,A -85,B 0,C 180,E1 2747.337,E2 2747.337} C_VEL
LIN {X 0,Y 68.897,Z 755.245,A -85,B 0,C 180,E1 2734.196,E2 2734.196} C_VEL
LIN {X 0,Y 82.448,Z 751.06,A -85,B 0,C 180,E1 2725.117,E2 2725.117} C_VEL
LIN {X 0,Y 97.138,Z 745.806,A -85,B 0,C 180,E1 2718.76,E2 2718.76} C_VEL
LIN {X 0,Y 112.39,Z 739.484,A -85,B 0,C 180,E1 2714.165,E2 2714.165} C_VEL
LIN {X 0,Y 130.072,Z 730.99,A -85,B 0,C 180,E1 2710.318,E2 2710.318} C_VEL
LIN {X 0,Y 150.127,Z 719.508,A -85,B 0,C 180,E1 2707.14,E2 2707.14} C_VEL
LIN {X 0,Y 165.653,Z 709.168,A -85,B 0,C 180,E1 2705.244,E2 2705.244} C_VEL
LIN {X 0,Y 179.767,Z 698.535,A -85,B 0,C 180,E1 2703.827,E2 2703.827} C_VEL
LIN {X 0,Y 193.443,Z 686.928,A -85,B 0,C 180,E1 2702.667,E2 2702.667} C_VEL
LIN {X 0,Y 206.541,Z 674.406,A -85,B 0,C 180,E1 2701.711,E2 2701.711} C_VEL
LIN {X 0,Y 219.473,Z 660.447,A -85,B 0,C 180,E1 2700.899,E2 2700.899} C_VEL
LIN {X 0,Y 234.363,Z 641.907,A -85,B 0,C 180,E1 2700.087,E2 2700.087} C_VEL
LIN {X 0,Y 245.981,Z 624.829,A -85,B 0,C 180,E1 2699.534,E2 2699.534} C_VEL
LIN {X 0,Y 255.466,Z 608.763,A -85,B 0,C 180,E1 2699.129,E2 2699.129} C_VEL
LIN {X 0,Y 263.491,Z 593.053,A -85,B 0,C 180,E1 2698.815,E2 2698.815} C_VEL
LIN {X 0,Y 270.519,Z 576.989,A -85,B 0,C 180,E1 2698.56,E2 2698.56} C_VEL
LIN {X 0,Y 276.795,Z 559.886,A -85,B 0,C 180,E1 2698.357,E2 2698.357} C_VEL
LIN {X 0,Y 277.991,Z 556.35,A -85,B 0,C 180,E1 2698.319,E2 2698.319} C_VEL
LIN {X 0,Y 280.303,Z 549.059,A -85,B 0,C 180,E1 2698.042,E2 2698.042} C_VEL
LIN {X 0,Y 285.12,Z 530.707,A -85,B 0,C 180,E1 2696.674,E2 2696.674} C_VEL
LIN {X 0,Y 286.776,Z 523.228,A -85,B 0,C 180,E1 2696.416,E2 2696.416} C_VEL
LIN {X 0,Y 289.948,Z 503.753,A -85,B 0,C 180,E1 2696.243,E2 2696.243} C_VEL
LIN {X 0,Y 290.385,Z 507.152,A -85,B 0,C 180,E1 2693.972,E2 2693.972} C_VEL
LIN {X 0,Y 290.886,Z 511.924,A -85,B 0,C 180,E1 2691.948,E2 2691.948} C_VEL
LIN {X 0,Y 291.614,Z 519.556,A -85,B 0,C 180,E1 2689.58,E2 2689.58} C_VEL
LIN {X 0,Y 294.469,Z 538.729,A -85,B 0,C 180,E1 2683.58,E2 2683.58} C_VEL
LIN {X 0,Y 299.442,Z 554.672,A -85,B 0,C 180,E1 2678.038,E2 2678.038} C_VEL
LIN {X 0,Y 306.764,Z 569.113,A -85,B 0,C 180,E1 2672.639,E2 2672.639} C_VEL
LIN {X 0,Y 320.536,Z 586.973,A -85,B 0,C 180,E1 2665.624,E2 2665.624} C_VEL
LIN {X 0,Y 341.029,Z 605.646,A -85,B 0,C 180,E1 2658.275,E2 2658.275} C_VEL
LIN {X 0,Y 360.303,Z 620.414,A -85,B 0,C 180,E1 2652.892,E2 2652.892} C_VEL
LIN {X 0,Y 372.778,Z 629.792,A -85,B 0,C 180,E1 2649.663,E2 2649.663} C_VEL
LIN {X 0,Y 381.683,Z 636.54,A -85,B 0,C 180,E1 2647.213,E2 2647.213} C_VEL
LIN {X 0,Y 389.588,Z 642.62,A -85,B 0,C 180,E1 2644.908,E2 2644.908} C_VEL
LIN {X 0,Y 396.555,Z 647.601,A -85,B 0,C 180,E1 2642.822,E2 2642.822} C_VEL
LIN {X 0,Y 404.463,Z 653.564,A -85,B 0,C 180,E1 2640.281,E2 2640.281} C_VEL
LIN {X 0,Y 413.135,Z 659.453,A -85,B 0,C 180,E1 2637.348,E2 2637.348} C_VEL
LIN {X 0,Y 421.08,Z 665.518,A -85,B 0,C 180,E1 2634.238,E2 2634.238} C_VEL
LIN {X 0,Y 428.191,Z 670.061,A -85,B 0,C 180,E1 2631.294,E2 2631.294} C_VEL
LIN {X 0,Y 433.287,Z 674.119,A -85,B 0,C 180,E1 2628.707,E2 2628.707} C_VEL
LIN {X 0,Y 438.812,Z 677.747,A -85,B 0,C 180,E1 2625.731,E2 2625.731} C_VEL
LIN {X 0,Y 443.323,Z 680.079,A -85,B 0,C 180,E1 2623.033,E2 2623.033} C_VEL
LIN {X 0,Y 446.377,Z 682.725,A -85,B 0,C 180,E1 2620.322,E2 2620.322} C_VEL
LIN {X 0,Y 448.818,Z 684.841,A -85,B 0,C 180,E1 2617.524,E2 2617.524} C_VEL
LIN {X 0,Y 450.576,Z 686.08,A -85,B 0,C 180,E1 2614.865,E2 2614.865} C_VEL
LIN {X 0,Y 451.574,Z 686.738,A -85,B 0,C 180,E1 2612.411,E2 2612.411} C_VEL
LIN {X 0,Y 451.886,Z 686.902,A -85,B 0,C 180,E1 2609.746,E2 2609.746} C_VEL
LIN {X 0,Y 451.5,Z 686.68,A -85,B 0,C 180,E1 2607.177,E2 2607.177} C_VEL
LIN {X 0,Y 450.283,Z 685.871,A -85,B 0,C 180,E1 2604.522,E2 2604.522} C_VEL
LIN {X 0,Y 448.273,Z 684.425,A -85,B 0,C 180,E1 2601.794,E2 2601.794} C_VEL
LIN {X 0,Y 445.679,Z 682.127,A -85,B 0,C 180,E1 2599.008,E2 2599.008} C_VEL
LIN {X 0,Y 443.117,Z 679.99,A -85,B 0,C 180,E1 2596.828,E2 2596.828} C_VEL
LIN {X 0,Y 438.834,Z 677.768,A -85,B 0,C 180,E1 2594.27,E2 2594.27} C_VEL
LIN {X 0,Y 433.287,Z 674.122,A -85,B 0,C 180,E1 2591.293,E2 2591.293} C_VEL
LIN {X 0,Y 428.039,Z 669.932,A -85,B 0,C 180,E1 2588.632,E2 2588.632} C_VEL
LIN {X 0,Y 421.032,Z 665.488,A -85,B 0,C 180,E1 2585.745,E2 2585.745} C_VEL
LIN {X 0,Y 413.055,Z 659.385,A -85,B 0,C 180,E1 2582.621,E2 2582.621} C_VEL
LIN {X 0,Y 404.305,Z 653.45,A -85,B 0,C 180,E1 2579.669,E2 2579.669} C_VEL
LIN {X 0,Y 396.429,Z 647.524,A -85,B 0,C 180,E1 2577.131,E2 2577.131} C_VEL
LIN {X 0,Y 386.851,Z 640.506,A -85,B 0,C 180,E1 2574.252,E2 2574.252} C_VEL
LIN {X 0,Y 377.506,Z 633.488,A -85,B 0,C 180,E1 2571.629,E2 2571.629} C_VEL
LIN {X 0,Y 369.002,Z 626.985,A -85,B 0,C 180,E1 2569.352,E2 2569.352} C_VEL
LIN {X 0,Y 354.888,Z 616.355,A -85,B 0,C 180,E1 2565.696,E2 2565.696} C_VEL
LIN {X 0,Y 335.313,Z 600.842,A -85,B 0,C 180,E1 2559.876,E2 2559.876} C_VEL
LIN {X 0,Y 317.484,Z 583.476,A -85,B 0,C 180,E1 2553.014,E2 2553.014} C_VEL
LIN {X 0,Y 304.794,Z 565.744,A -85,B 0,C 180,E1 2546.078,E2 2546.078} C_VEL
LIN {X 0,Y 297.868,Z 550.607,A -85,B 0,C 180,E1 2540.489,E2 2540.489} C_VEL
LIN {X 0,Y 293.304,Z 532.885,A -85,B 0,C 180,E1 2534.525,E2 2534.525} C_VEL
LIN {X 0,Y 291.246,Z 515.352,A -85,B 0,C 180,E1 2529.186,E2 2529.186} C_VEL
LIN {X 0,Y 290.621,Z 508.99,A -85,B 0,C 180,E1 2526.916,E2 2526.916} C_VEL
LIN {X 0,Y 290.062,Z 504.405,A -85,B 0,C 180,E1 2524.349,E2 2524.349} C_VEL
LIN {X 0,Y 289.92,Z 503.939,A -85,B 0,C 180,E1 2523.744,E2 2523.744} C_VEL
LIN {X 0,Y 286.106,Z 526.348,A -85,B 0,C 180,E1 2523.559,E2 2523.559} C_VEL
LIN {X 0,Y 281.649,Z 544.861,A -85,B 0,C 180,E1 2523.416,E2 2523.416} C_VEL
LIN {X 0,Y 276.132,Z 562.692,A -85,B 0,C 180,E1 2523.274,E2 2523.274} C_VEL
LIN {X 0,Y 269.326,Z 580.547,A -85,B 0,C 180,E1 2523.095,E2 2523.095} C_VEL
LIN {X 0,Y 259.243,Z 602.157,A -85,B 0,C 180,E1 2522.789,E2 2522.789} C_VEL
LIN {X 0,Y 248.662,Z 620.685,A -85,B 0,C 180,E1 2522.432,E2 2522.432} C_VEL
LIN {X 0,Y 238.594,Z 635.942,A -85,B 0,C 180,E1 2522.054,E2 2522.054} C_VEL
LIN {X 0,Y 228.033,Z 650.01,A -85,B 0,C 180,E1 2521.61,E2 2521.61} C_VEL
LIN {X 0,Y 216.371,Z 663.758,A -85,B 0,C 180,E1 2521.059,E2 2521.059} C_VEL
LIN {X 0,Y 203.454,Z 677.224,A -85,B 0,C 180,E1 2520.367,E2 2520.367} C_VEL
LIN {X 0,Y 186.967,Z 692.331,A -85,B 0,C 180,E1 2519.314,E2 2519.314} C_VEL
LIN {X 0,Y 169.069,Z 706.186,A -85,B 0,C 180,E1 2517.925,E2 2517.925} C_VEL
LIN {X 0,Y 154.248,Z 716.236,A -85,B 0,C 180,E1 2516.507,E2 2516.507} C_VEL
LIN {X 0,Y 139.544,Z 725.027,A -85,B 0,C 180,E1 2514.779,E2 2514.779} C_VEL
LIN {X 0,Y 124.036,Z 733.156,A -85,B 0,C 180,E1 2512.48,E2 2512.48} C_VEL
LIN {X 0,Y 108.784,Z 740.105,A -85,B 0,C 180,E1 2509.532,E2 2509.532} C_VEL
LIN {X 0,Y 92.995,Z 746.297,A -85,B 0,C 180,E1 2505.364,E2 2505.364} C_VEL
LIN {X 0,Y 77.018,Z 751.606,A -85,B 0,C 180,E1 2499.165,E2 2499.165} C_VEL
LIN {X 0,Y 58.618,Z 756.661,A -85,B 0,C 180,E1 2486.69,E2 2486.69} C_VEL
LIN {X 0,Y 45.771,Z 759.476,A -85,B 0,C 180,E1 2467.704,E2 2467.704} C_VEL
LIN {X 0,Y 40.44,Z 760.684,A -85,B 0,C 180,E1 2445.355,E2 2445.355} C_VEL
LIN {X 0,Y 40.001,Z 760.987,A -85,B 0,C 180,E1 2428.568,E2 2428.568} C_VEL
LIN {X 0,Y 42.261,Z 760.294,A -85,B 0,C 180,E1 2403.29,E2 2403.29} C_VEL
LIN {X 0,Y 51.839,Z 758.163,A -85,B 0,C 180,E1 2381.224,E2 2381.224} C_VEL
LIN {X 0,Y 64.66,Z 755.066,A -85,B 0,C 180,E1 2368.198,E2 2368.198} C_VEL
LIN {X 0,Y 78.742,Z 751.063,A -85,B 0,C 180,E1 2360.025,E2 2360.025} C_VEL
LIN {X 0,Y 93.909,Z 745.962,A -85,B 0,C 180,E1 2354.353,E2 2354.353} C_VEL
LIN {X 0,Y 109.728,Z 739.705,A -85,B 0,C 180,E1 2350.26,E2 2350.26} C_VEL
LIN {X 0,Y 125.963,Z 732.218,A -85,B 0,C 180,E1 2347.201,E2 2347.201} C_VEL
LIN {X 0,Y 145.411,Z 721.775,A -85,B 0,C 180,E1 2344.492,E2 2344.492} C_VEL
LIN {X 0,Y 164.118,Z 709.692,A -85,B 0,C 180,E1 2342.52,E2 2342.52} C_VEL
LIN {X 0,Y 178.999,Z 698.682,A -85,B 0,C 180,E1 2341.266,E2 2341.266} C_VEL
LIN {X 0,Y 192.955,Z 687,A -85,B 0,C 180,E1 2340.279,E2 2340.279} C_VEL
LIN {X 0,Y 205.957,Z 674.729,A -85,B 0,C 180,E1 2339.49,E2 2339.49} C_VEL
LIN {X 0,Y 218.491,Z 661.392,A -85,B 0,C 180,E1 2338.835,E2 2338.835} C_VEL
LIN {X 0,Y 232.558,Z 644.344,A -85,B 0,C 180,E1 2338.195,E2 2338.195} C_VEL
LIN {X 0,Y 245.87,Z 625.149,A -85,B 0,C 180,E1 2337.669,E2 2337.669} C_VEL
LIN {X 0,Y 255.211,Z 609.513,A -85,B 0,C 180,E1 2337.343,E2 2337.343} C_VEL
LIN {X 0,Y 263.78,Z 592.885,A -85,B 0,C 180,E1 2337.069,E2 2337.069} C_VEL
LIN {X 0,Y 271.344,Z 575.575,A -85,B 0,C 180,E1 2336.848,E2 2336.848} C_VEL
LIN {X 0,Y 278.402,Z 556.006,A -85,B 0,C 180,E1 2336.667,E2 2336.667} C_VEL
LIN {X 0,Y 284.808,Z 532.389,A -85,B 0,C 180,E1 2336.489,E2 2336.489} C_VEL
LIN {X 0,Y 286.776,Z 523.228,A -85,B 0,C 180,E1 2336.416,E2 2336.416} C_VEL
LIN {X 0,Y 287.307,Z 521.047,A -85,B 0,C 180,E1 2336.194,E2 2336.194} C_VEL
LIN {X 0,Y 287.888,Z 519.3,A -85,B 0,C 180,E1 2335.576,E2 2335.576} C_VEL
LIN {X 0,Y 288.432,Z 518.708,A -85,B 0,C 180,E1 2334.563,E2 2334.563} C_VEL
LIN {X 0,Y 288.818,Z 519.86,A -85,B 0,C 180,E1 2333.332,E2 2333.332} C_VEL
LIN {X 0,Y 289.31,Z 523.93,A -85,B 0,C 180,E1 2331.267,E2 2331.267} C_VEL
LIN {X 0,Y 289.637,Z 528.417,A -85,B 0,C 180,E1 2329.701,E2 2329.701} C_VEL
LIN {X 0,Y 291.595,Z 545.274,A -85,B 0,C 180,E1 2324.283,E2 2324.283} C_VEL
LIN {X 0,Y 295.511,Z 560.086,A -85,B 0,C 180,E1 2319.026,E2 2319.026} C_VEL
LIN {X 0,Y 300.822,Z 572.233,A -85,B 0,C 180,E1 2314.399,E2 2314.399} C_VEL
LIN {X 0,Y 311.465,Z 588.136,A -85,B 0,C 180,E1 2308.015,E2 2308.015} C_VEL
LIN {X 0,Y 328.79,Z 605.836,A -85,B 0,C 180,E1 2300.761,E2 2300.761} C_VEL
LIN {X 0,Y 348.955,Z 621.9,A -85,B 0,C 180,E1 2294.481,E2 2294.481} C_VEL
LIN {X 0,Y 365.679,Z 634.326,A -85,B 0,C 180,E1 2290.038,E2 2290.038} C_VEL
LIN {X 0,Y 374.162,Z 640.883,A -85,B 0,C 180,E1 2287.719,E2 2287.719} C_VEL
LIN {X 0,Y 381.474,Z 646.403,A -85,B 0,C 180,E1 2285.654,E2 2285.654} C_VEL
LIN {X 0,Y 389.165,Z 652.131,A -85,B 0,C 180,E1 2283.351,E2 2283.351} C_VEL
LIN {X 0,Y 395.669,Z 656.867,A -85,B 0,C 180,E1 2281.333,E2 2281.333} C_VEL
LIN {X 0,Y 404.05,Z 662.928,A -85,B 0,C 180,E1 2278.537,E2 2278.537} C_VEL
LIN {X 0,Y 409.169,Z 666.519,A -85,B 0,C 180,E1 2276.717,E2 2276.717} C_VEL
LIN {X 0,Y 416.196,Z 671.739,A -85,B 0,C 180,E1 2273.951,E2 2273.951} C_VEL
LIN {X 0,Y 422.885,Z 676.039,A -85,B 0,C 180,E1 2271.205,E2 2271.205} C_VEL
LIN {X 0,Y 428.748,Z 680.634,A -85,B 0,C 180,E1 2268.208,E2 2268.208} C_VEL
LIN {X 0,Y 433.731,Z 683.817,A -85,B 0,C 180,E1 2265.5,E2 2265.5} C_VEL
LIN {X 0,Y 438.453,Z 686.254,A -85,B 0,C 180,E1 2262.644,E2 2262.644} C_VEL
LIN {X 0,Y 441.488,Z 689.089,A -85,B 0,C 180,E1 2259.778,E2 2259.778} C_VEL
LIN {X 0,Y 443.789,Z 691.002,A -85,B 0,C 180,E1 2256.987,E2 2256.987} C_VEL
LIN {X 0,Y 445.276,Z 692.053,A -85,B 0,C 180,E1 2254.417,E2 2254.417} C_VEL
LIN {X 0,Y 446.212,Z 692.632,A -85,B 0,C 180,E1 2251.669,E2 2251.669} C_VEL
LIN {X 0,Y 446.332,Z 692.685,A -85,B 0,C 180,E1 2249.358,E2 2249.358} C_VEL
LIN {X 0,Y 445.807,Z 692.385,A -85,B 0,C 180,E1 2246.786,E2 2246.786} C_VEL
LIN {X 0,Y 444.417,Z 691.431,A -85,B 0,C 180,E1 2243.965,E2 2243.965} C_VEL
LIN {X 0,Y 442.263,Z 689.807,A -85,B 0,C 180,E1 2241.113,E2 2241.113} C_VEL
LIN {X 0,Y 439.654,Z 687.459,A -85,B 0,C 180,E1 2238.457,E2 2238.457} C_VEL
LIN {X 0,Y 437.556,Z 685.808,A -85,B 0,C 180,E1 2236.777,E2 2236.777} C_VEL
LIN {X 0,Y 432.662,Z 683.203,A -85,B 0,C 180,E1 2233.902,E2 2233.902} C_VEL
LIN {X 0,Y 427.539,Z 679.752,A -85,B 0,C 180,E1 2231.174,E2 2231.174} C_VEL
LIN {X 0,Y 421.805,Z 675.23,A -85,B 0,C 180,E1 2228.3,E2 2228.3} C_VEL
LIN {X 0,Y 413.982,Z 670.22,A -85,B 0,C 180,E1 2225.153,E2 2225.153} C_VEL
LIN {X 0,Y 406.555,Z 664.549,A -85,B 0,C 180,E1 2222.3,E2 2222.3} C_VEL
LIN {X 0,Y 397.624,Z 658.38,A -85,B 0,C 180,E1 2219.309,E2 2219.309} C_VEL
LIN {X 0,Y 390.651,Z 653.152,A -85,B 0,C 180,E1 2217.091,E2 2217.091} C_VEL
LIN {X 0,Y 382.822,Z 647.456,A -85,B 0,C 180,E1 2214.75,E2 2214.75} C_VEL
LIN {X 0,Y 375.237,Z 641.678,A -85,B 0,C 180,E1 2212.569,E2 2212.569} C_VEL
LIN {X 0,Y 365.164,Z 633.979,A -85,B 0,C 180,E1 2209.814,E2 2209.814} C_VEL
LIN {X 0,Y 348.424,Z 621.51,A -85,B 0,C 180,E1 2205.373,E2 2205.373} C_VEL
LIN {X 0,Y 328.79,Z 605.837,A -85,B 0,C 180,E1 2199.239,E2 2199.239} C_VEL
LIN {X 0,Y 311.464,Z 588.136,A -85,B 0,C 180,E1 2191.985,E2 2191.985} C_VEL
LIN {X 0,Y 300.316,Z 571.307,A -85,B 0,C 180,E1 2185.225,E2 2185.225} C_VEL
LIN {X 0,Y 294.321,Z 556.536,A -85,B 0,C 180,E1 2179.653,E2 2179.653} C_VEL
LIN {X 0,Y 290.646,Z 538.807,A -85,B 0,C 180,E1 2173.58,E2 2173.58} C_VEL
LIN {X 0,Y 289.362,Z 519.059,A -85,B 0,C 180,E1 2167.4,E2 2167.4} C_VEL
LIN {X 0,Y 289.021,Z 514.497,A -85,B 0,C 180,E1 2165.459,E2 2165.459} C_VEL
LIN {X 0,Y 288.95,Z 514.322,A -85,B 0,C 180,E1 2165.243,E2 2165.243} C_VEL
LIN {X 0,Y 283.975,Z 538.434,A -85,B 0,C 180,E1 2165.077,E2 2165.077} C_VEL
LIN {X 0,Y 277.812,Z 559.28,A -85,B 0,C 180,E1 2164.955,E2 2164.955} C_VEL
LIN {X 0,Y 271.397,Z 576.647,A -85,B 0,C 180,E1 2164.831,E2 2164.831} C_VEL
LIN {X 0,Y 263.807,Z 593.778,A -85,B 0,C 180,E1 2164.66,E2 2164.66} C_VEL
LIN {X 0,Y 254.442,Z 611.649,A -85,B 0,C 180,E1 2164.425,E2 2164.425} C_VEL
LIN {X 0,Y 240.984,Z 633.01,A -85,B 0,C 180,E1 2164.045,E2 2164.045} C_VEL
LIN {X 0,Y 229.414,Z 648.579,A -85,B 0,C 180,E1 2163.672,E2 2163.672} C_VEL
LIN {X 0,Y 217.795,Z 662.34,A -85,B 0,C 180,E1 2163.245,E2 2163.245} C_VEL
LIN {X 0,Y 205.18,Z 675.555,A -85,B 0,C 180,E1 2162.717,E2 2162.717} C_VEL
LIN {X 0,Y 192.079,Z 687.715,A -85,B 0,C 180,E1 2162.079,E2 2162.079} C_VEL
LIN {X 0,Y 176.996,Z 700.088,A -85,B 0,C 180,E1 2161.212,E2 2161.212} C_VEL
LIN {X 0,Y 156.962,Z 714.202,A -85,B 0,C 180,E1 2159.784,E2 2159.784} C_VEL
LIN {X 0,Y 140.032,Z 724.307,A -85,B 0,C 180,E1 2158.234,E2 2158.234} C_VEL
LIN {X 0,Y 123.498,Z 732.851,A -85,B 0,C 180,E1 2156.286,E2 2156.286} C_VEL
LIN {X 0,Y 107.599,Z 739.927,A -85,B 0,C 180,E1 2153.817,E2 2153.817} C_VEL
LIN {X 0,Y 91.272,Z 746.118,A -85,B 0,C 180,E1 2150.337,E2 2150.337} C_VEL
LIN {X 0,Y 74.503,Z 751.428,A -85,B 0,C 180,E1 2145.053,E2 2145.053} C_VEL
LIN {X 0,Y 54.565,Z 756.483,A -85,B 0,C 180,E1 2133.869,E2 2133.869} C_VEL
LIN {X 0,Y 39.653,Z 759.299,A -85,B 0,C 180,E1 2114.906,E2 2114.906} C_VEL
LIN {X 0,Y 32.621,Z 760.525,A -85,B 0,C 180,E1 2088.156,E2 2088.156} C_VEL
LIN {X 0,Y 31.992,Z 760.812,A -85,B 0,C 180,E1 2068.209,E2 2068.209} C_VEL
LIN {X 0,Y 35.622,Z 760.026,A -85,B 0,C 180,E1 2035.853,E2 2035.853} C_VEL
LIN {X 0,Y 47.601,Z 757.835,A -85,B 0,C 180,E1 2012.848,E2 2012.848} C_VEL
LIN {X 0,Y 62.082,Z 754.678,A -85,B 0,C 180,E1 2000.931,E2 2000.931} C_VEL
LIN {X 0,Y 77.247,Z 750.613,A -85,B 0,C 180,E1 1993.911,E2 1993.911} C_VEL
LIN {X 0,Y 93.174,Z 745.449,A -85,B 0,C 180,E1 1989.191,E2 1989.191} C_VEL
LIN {X 0,Y 110.202,Z 738.854,A -85,B 0,C 180,E1 1985.728,E2 1985.728} C_VEL
LIN {X 0,Y 130.132,Z 729.693,A -85,B 0,C 180,E1 1982.874,E2 1982.874} C_VEL
LIN {X 0,Y 149.978,Z 718.533,A -85,B 0,C 180,E1 1980.811,E2 1980.811} C_VEL
LIN {X 0,Y 164.963,Z 708.813,A -85,B 0,C 180,E1 1979.601,E2 1979.601} C_VEL
LIN {X 0,Y 179.005,Z 698.507,A -85,B 0,C 180,E1 1978.663,E2 1978.663} C_VEL
LIN {X 0,Y 193.086,Z 686.826,A -85,B 0,C 180,E1 1977.87,E2 1977.87} C_VEL
LIN {X 0,Y 206.499,Z 674.249,A -85,B 0,C 180,E1 1977.225,E2 1977.225} C_VEL
LIN {X 0,Y 220.32,Z 659.54,A -85,B 0,C 180,E1 1976.659,E2 1976.659} C_VEL
LIN {X 0,Y 235.897,Z 640.156,A -85,B 0,C 180,E1 1976.111,E2 1976.111} C_VEL
LIN {X 0,Y 247.111,Z 623.733,A -85,B 0,C 180,E1 1975.773,E2 1975.773} C_VEL
LIN {X 0,Y 256.723,Z 607.504,A -85,B 0,C 180,E1 1975.513,E2 1975.513} C_VEL
LIN {X 0,Y 265.324,Z 590.594,A -85,B 0,C 180,E1 1975.306,E2 1975.306} C_VEL
LIN {X 0,Y 273.925,Z 570.431,A -85,B 0,C 180,E1 1975.122,E2 1975.122} C_VEL
LIN {X 0,Y 281.319,Z 548.029,A -85,B 0,C 180,E1 1974.978,E2 1974.978} C_VEL
LIN {X 0,Y 286.143,Z 528.839,A -85,B 0,C 180,E1 1974.859,E2 1974.859} C_VEL
LIN {X 0,Y 288.945,Z 514.144,A -85,B 0,C 180,E1 1974.739,E2 1974.739} C_VEL
LIN {X 0,Y 289.295,Z 518.245,A -85,B 0,C 180,E1 1972.902,E2 1972.902} C_VEL
LIN {X 0,Y 289.5,Z 524.515,A -85,B 0,C 180,E1 1970.858,E2 1970.858} C_VEL
LIN {X 0,Y 289.637,Z 528.417,A -85,B 0,C 180,E1 1969.701,E2 1969.701} C_VEL
LIN {X 0,Y 289.701,Z 533.393,A -85,B 0,C 180,E1 1968.518,E2 1968.518} C_VEL
LIN {X 0,Y 288.692,Z 548.265,A -85,B 0,C 180,E1 1965.843,E2 1965.843} C_VEL
LIN {X 0,Y 288.88,Z 552.893,A -85,B 0,C 180,E1 1964.615,E2 1964.615} C_VEL
LIN {X 0,Y 293.04,Z 569.896,A -85,B 0,C 180,E1 1958.376,E2 1958.376} C_VEL
LIN {X 0,Y 301.231,Z 586.541,A -85,B 0,C 180,E1 1951.662,E2 1951.662} C_VEL
LIN {X 0,Y 315.299,Z 604.052,A -85,B 0,C 180,E1 1944.265,E2 1944.265} C_VEL
LIN {X 0,Y 336.869,Z 622.629,A -85,B 0,C 180,E1 1936.479,E2 1936.479} C_VEL
LIN {X 0,Y 352.367,Z 634.411,A -85,B 0,C 180,E1 1931.973,E2 1931.973} C_VEL
LIN {X 0,Y 363.828,Z 642.989,A -85,B 0,C 180,E1 1928.944,E2 1928.944} C_VEL
LIN {X 0,Y 373.913,Z 650.495,A -85,B 0,C 180,E1 1926.139,E2 1926.139} C_VEL
LIN {X 0,Y 382.143,Z 656.81,A -85,B 0,C 180,E1 1923.685,E2 1923.685} C_VEL
LIN {X 0,Y 388.918,Z 661.641,A -85,B 0,C 180,E1 1921.628,E2 1921.628} C_VEL
LIN {X 0,Y 397.274,Z 667.825,A -85,B 0,C 180,E1 1918.851,E2 1918.851} C_VEL
LIN {X 0,Y 403.2,Z 671.906,A -85,B 0,C 180,E1 1916.777,E2 1916.777} C_VEL
LIN {X 0,Y 409.861,Z 676.922,A -85,B 0,C 180,E1 1914.16,E2 1914.16} C_VEL
LIN {X 0,Y 416.356,Z 681.002,A -85,B 0,C 180,E1 1911.554,E2 1911.554} C_VEL
LIN {X 0,Y 422.49,Z 685.855,A -85,B 0,C 180,E1 1908.487,E2 1908.487} C_VEL
LIN {X 0,Y 427.799,Z 689.299,A -85,B 0,C 180,E1 1905.59,E2 1905.59} C_VEL
LIN {X 0,Y 432.734,Z 691.882,A -85,B 0,C 180,E1 1902.679,E2 1902.679} C_VEL
LIN {X 0,Y 435.631,Z 694.553,A -85,B 0,C 180,E1 1899.911,E2 1899.911} C_VEL
LIN {X 0,Y 437.983,Z 696.533,A -85,B 0,C 180,E1 1897.08,E2 1897.08} C_VEL
LIN {X 0,Y 439.493,Z 697.597,A -85,B 0,C 180,E1 1894.567,E2 1894.567} C_VEL
LIN {X 0,Y 440.505,Z 698.241,A -85,B 0,C 180,E1 1891.821,E2 1891.821} C_VEL
LIN {X 0,Y 440.652,Z 698.313,A -85,B 0,C 180,E1 1889.48,E2 1889.48} C_VEL
LIN {X 0,Y 440.206,Z 698.055,A -85,B 0,C 180,E1 1887.006,E2 1887.006} C_VEL
LIN {X 0,Y 438.883,Z 697.156,A -85,B 0,C 180,E1 1884.248,E2 1884.248} C_VEL
LIN {X 0,Y 436.788,Z 695.606,A -85,B 0,C 180,E1 1881.444,E2 1881.444} C_VEL
LIN {X 0,Y 434.233,Z 693.332,A -85,B 0,C 180,E1 1878.714,E2 1878.714} C_VEL
